// TwinCAT 3 PLC project BROTLibTests
// Title: BROTLibTests
// Company: BROT
// ProjectVersion: 0.1.0
// ProgramVersion: 3.1.4024.66
// libraries:
//   BROTLib, * (BROT)
//   Tc2_MC2, * (Beckhoff Automation GmbH)
//   Tc2_MC2_Drive, * (Beckhoff Automation GmbH)
//   Tc2_NC, * (Beckhoff Automation GmbH)
//   Tc2_Standard, * (Beckhoff Automation GmbH)
//   Tc2_System, * (Beckhoff Automation GmbH)
//   Tc2_Utilities, * (Beckhoff Automation GmbH)
//   Tc3_Module, * (Beckhoff Automation GmbH)
//   TcUnit, * (www.tcunit.org)
// project tree:
//   / PlcTask.TcTTO
//   POUs/ FB_Axis_Tests.TcPOU, FB_Blink_Tests.TcPOU, FB_AstroClockSync_Tests.TcPOU, FB_InfluxLineProtocol_Tests.TcPOU, FB_InfluxMessage_Tests.TcPOU, FB_TelescopeStub.TcPOU, FB_Comm_MQTT_Influx_Tests.TcPOU, FB_BlinkTimingProbe.TcPOU, FB_EscapeInfluxString_Tests.TcPOU, F_SetpointEnableExecute_Tests.TcPOU, FB_InfoConnection_Tests.TcPOU, FB_IsNumericValue_Tests.TcPOU, FB_PointingModel_Tests.TcPOU, FB_Tracking_Tests.TcPOU, FB_YREAL_Tests.TcPOU, MAIN.TcPOU
// real-time tasks:
//   TASK PlcTask: cycle T#10ms, priority 20, ADS port 350

CONFIGURATION BROTLibTests
    RESOURCE PLC ON TwinCAT3
        TASK PlcTask(INTERVAL := T#10ms, PRIORITY := 20);
        PROGRAM MAIN WITH PlcTask : MAIN;
    END_RESOURCE
END_CONFIGURATION

// ---- POUs/MAIN.TcPOU
PROGRAM MAIN
VAR
	// TcUnit finds every FB_TestSuite instance by itself; it is enough to declare them here.
	fbIsNumericValueTests	: FB_IsNumericValue_Tests;
	fbEscapeInfluxTests		: FB_EscapeInfluxString_Tests;
	fbYRealTests			: FB_YREAL_Tests;
	fbTrackingTests			: FB_Tracking_Tests;
	fbPointingModelTests	: FB_PointingModel_Tests;
	fbBlinkTests			: FB_Blink_Tests;
	fbAxisTests				: FB_Axis_Tests;
	fbAstroClockSyncTests	: FB_AstroClockSync_Tests;
	fbInfluxLineProtocolTests	: FB_InfluxLineProtocol_Tests;
	fbInfluxMessageTests		: FB_InfluxMessage_Tests;
	fbCommMqttInfluxTests		: FB_Comm_MQTT_Influx_Tests;
	fbInfoConnectionTests		: FB_InfoConnection_Tests;
	fbSetpointEnableTests		: F_SetpointEnableExecute_Tests;
END_VAR

TcUnit.RUN();

END_PROGRAM

// ---- POUs/FB_IsNumericValue_Tests.TcPOU
// Tests for BROTLib.F_IsNumericValue, which decides whether an Influx field value is written as a number.
FUNCTION_BLOCK FB_IsNumericValue_Tests EXTENDS TcUnit.FB_TestSuite
VAR
END_VAR

Accepts_Plain_Numbers();
Accepts_Signs_And_Exponents();
Rejects_Malformed_Numbers();
Rejects_Non_Numeric_Text();

// Asserts F_IsNumericValue(sValue) = bExpected; the failure message names the offending input.
METHOD PRIVATE Check
VAR_INPUT
	sValue		: STRING(255);
	bExpected	: BOOL;
END_VAR
AssertEquals_BOOL(
	Expected := bExpected,
	Actual := BROTLib.F_IsNumericValue(sValue := sValue),
	Message := CONCAT('F_IsNumericValue on input: ', sValue));
END_METHOD

METHOD PRIVATE Accepts_Plain_Numbers
VAR
	aCases	: ARRAY[1..6] OF STRING(255) := ['0', '15', '15.5', '007', '0.001', '123456789012345678'];
	i		: INT;
END_VAR
TEST('Accepts_Plain_Numbers');
FOR i := 1 TO 6 DO
	Check(sValue := aCases[i], bExpected := TRUE);
END_FOR
TEST_FINISHED();
END_METHOD

METHOD PRIVATE Accepts_Signs_And_Exponents
VAR
	aCases	: ARRAY[1..8] OF STRING(255) := ['-3', '+7', '-0.5', '1e5', '1E-05', '1.0E-5', '-1.5e+3', '2.5E+10'];
	i		: INT;
END_VAR
TEST('Accepts_Signs_And_Exponents');
FOR i := 1 TO 8 DO
	Check(sValue := aCases[i], bExpected := TRUE);
END_FOR
TEST_FINISHED();
END_METHOD

METHOD PRIVATE Rejects_Malformed_Numbers
VAR
	aCases	: ARRAY[1..14] OF STRING(255) := ['', '-', '+', '.', 'e5', '1e', '1e+', '1.5.2', '1e5.5', '--1', '+-1', '1-1', '1e5e5', '1e--5'];
	i		: INT;
END_VAR
TEST('Rejects_Malformed_Numbers');
FOR i := 1 TO 14 DO
	Check(sValue := aCases[i], bExpected := FALSE);
END_FOR
TEST_FINISHED();
END_METHOD

METHOD PRIVATE Rejects_Non_Numeric_Text
VAR
	aCases	: ARRAY[1..9] OF STRING(255) := ['NaN', 'TRUE', 'abc', '12a', '50cm', ' 1', '1 ', '1,5', '0x1F'];
	i		: INT;
END_VAR
TEST('Rejects_Non_Numeric_Text');
FOR i := 1 TO 9 DO
	Check(sValue := aCases[i], bExpected := FALSE);
END_FOR
TEST_FINISHED();
END_METHOD

END_FUNCTION_BLOCK

// ---- POUs/FB_EscapeInfluxString_Tests.TcPOU
// Tests for BROTLib.F_EscapeInfluxString: inside a quoted InfluxDB string field only " and \ need escaping.
FUNCTION_BLOCK FB_EscapeInfluxString_Tests EXTENDS TcUnit.FB_TestSuite
VAR
END_VAR

Leaves_Plain_Text_Unchanged();
Escapes_Double_Quotes();
Escapes_Backslashes();
Doubles_Length_Of_All_Quote_Input();

METHOD PRIVATE Check
VAR_INPUT
	sInput		: STRING(255);
	sExpected	: STRING(255);
END_VAR
AssertEquals_STRING(
	Expected := sExpected,
	Actual := BROTLib.F_EscapeInfluxString(sValue := sInput),
	Message := CONCAT('F_EscapeInfluxString on input: ', sInput));
END_METHOD

METHOD PRIVATE Leaves_Plain_Text_Unchanged
VAR
END_VAR
TEST('Leaves_Plain_Text_Unchanged');
Check(sInput := '', sExpected := '');
Check(sInput := 'plain text', sExpected := 'plain text');
Check(sInput := 'a,b=c d', sExpected := 'a,b=c d');
Check(sInput := 'temp 21.5 C', sExpected := 'temp 21.5 C');
TEST_FINISHED();
END_METHOD

METHOD PRIVATE Escapes_Double_Quotes
VAR
END_VAR
TEST('Escapes_Double_Quotes');
Check(sInput := '"', sExpected := '\"');
Check(sInput := 'say "hi"', sExpected := 'say \"hi\"');
Check(sInput := '""', sExpected := '\"\"');
TEST_FINISHED();
END_METHOD

METHOD PRIVATE Escapes_Backslashes
VAR
END_VAR
TEST('Escapes_Backslashes');
Check(sInput := '\', sExpected := '\\');
Check(sInput := 'C:\temp', sExpected := 'C:\\temp');
// a backslash followed by a quote: both characters are escaped independently
Check(sInput := '\"', sExpected := '\\\"');
TEST_FINISHED();
END_METHOD

METHOD PRIVATE Doubles_Length_Of_All_Quote_Input
VAR
	sInput	: STRING(255);
	sOut	: STRING(255);
	i		: INT;
END_VAR
TEST('Doubles_Length_Of_All_Quote_Input');
sInput := '';
FOR i := 1 TO 100 DO
	sInput := CONCAT(sInput, '"');
END_FOR
sOut := BROTLib.F_EscapeInfluxString(sValue := sInput);
AssertEquals_INT(Expected := 200, Actual := LEN(sOut), Message := '100 quotes must become 100 escaped pairs');
AssertEquals_STRING(Expected := '\"\"', Actual := LEFT(sOut, 4), Message := 'every quote is preceded by one backslash');
TEST_FINISHED();
END_METHOD

END_FUNCTION_BLOCK

// ---- POUs/FB_YREAL_Tests.TcPOU
// Tests for BROTLib.F_YREAL, the linear scaling helper.
FUNCTION_BLOCK FB_YREAL_Tests EXTENDS TcUnit.FB_TestSuite
VAR
END_VAR

Default_Range_Maps_Raw_To_Unit();
Scales_To_Engineering_Range();
Clamps_Unless_Cut_Is_False();
Zero_Width_Input_Range_Returns_Zero();
Inverted_Output_Range_Maps_Correctly();

METHOD PRIVATE CheckNear
VAR_INPUT
	fExpected	: REAL;
	fActual		: REAL;
	fDelta		: REAL;
	sName		: STRING(255);
END_VAR
AssertEquals_REAL(Expected := fExpected, Actual := fActual, Delta := fDelta, Message := sName);
END_METHOD

METHOD PRIVATE Default_Range_Maps_Raw_To_Unit
VAR
END_VAR
TEST('Default_Range_Maps_Raw_To_Unit');
// defaults: 0..32767 -> 0..1
CheckNear(0.0, BROTLib.F_YREAL(fX := 0.0, fXmin := 0.0, fXmax := 32767.0, fYmin := 0.0, fYmax := 1.0, cut := TRUE), 1.0E-6, 'raw 0 -> 0');
CheckNear(1.0, BROTLib.F_YREAL(fX := 32767.0, fXmin := 0.0, fXmax := 32767.0, fYmin := 0.0, fYmax := 1.0, cut := TRUE), 1.0E-6, 'raw 32767 -> 1');
CheckNear(0.5, BROTLib.F_YREAL(fX := 16383.5, fXmin := 0.0, fXmax := 32767.0, fYmin := 0.0, fYmax := 1.0, cut := TRUE), 1.0E-6, 'raw mid-scale -> 0.5');
TEST_FINISHED();
END_METHOD

METHOD PRIVATE Scales_To_Engineering_Range
VAR
END_VAR
TEST('Scales_To_Engineering_Range');
// a 4..20 mA style input
CheckNear(4.0, BROTLib.F_YREAL(fX := 0.0, fXmin := 0.0, fXmax := 32767.0, fYmin := 4.0, fYmax := 20.0, cut := TRUE), 1.0E-5, '4..20: raw 0 -> 4');
CheckNear(20.0, BROTLib.F_YREAL(fX := 32767.0, fXmin := 0.0, fXmax := 32767.0, fYmin := 4.0, fYmax := 20.0, cut := TRUE), 1.0E-5, '4..20: raw 32767 -> 20');
CheckNear(12.0, BROTLib.F_YREAL(fX := 16383.5, fXmin := 0.0, fXmax := 32767.0, fYmin := 4.0, fYmax := 20.0, cut := TRUE), 1.0E-4, '4..20: mid-scale -> 12');
// symmetric ranges on both sides
CheckNear(0.0, BROTLib.F_YREAL(fX := 0.0, fXmin := -10.0, fXmax := 10.0, fYmin := -1.0, fYmax := 1.0, cut := TRUE), 1.0E-6, '-10..10 -> -1..1: 0 -> 0');
CheckNear(0.5, BROTLib.F_YREAL(fX := 5.0, fXmin := -10.0, fXmax := 10.0, fYmin := -1.0, fYmax := 1.0, cut := TRUE), 1.0E-6, '-10..10 -> -1..1: 5 -> 0.5');
CheckNear(-1.0, BROTLib.F_YREAL(fX := -10.0, fXmin := -10.0, fXmax := 10.0, fYmin := -1.0, fYmax := 1.0, cut := TRUE), 1.0E-6, '-10..10 -> -1..1: -10 -> -1');
TEST_FINISHED();
END_METHOD

METHOD PRIVATE Clamps_Unless_Cut_Is_False
VAR
END_VAR
TEST('Clamps_Unless_Cut_Is_False');
// cut defaults to TRUE
CheckNear(1.0, BROTLib.F_YREAL(fX := 40000.0, fXmin := 0.0, fXmax := 32767.0, fYmin := 0.0, fYmax := 1.0, cut := TRUE), 1.0E-6, 'above range is clamped to the maximum');
CheckNear(0.0, BROTLib.F_YREAL(fX := -100.0, fXmin := 0.0, fXmax := 32767.0, fYmin := 0.0, fYmax := 1.0, cut := TRUE), 1.0E-6, 'below range is clamped to the minimum');
CheckNear(20.0, BROTLib.F_YREAL(fX := 40000.0, fXmin := 0.0, fXmax := 32767.0, fYmin := 4.0, fYmax := 20.0, cut := TRUE), 1.0E-5, 'clamping works with an offset range');
// cut = FALSE extrapolates linearly
CheckNear(2.0, BROTLib.F_YREAL(fX := 65534.0, fXmin := 0.0, fXmax := 32767.0, fYmin := 0.0, fYmax := 1.0, cut := FALSE), 1.0E-5, 'unclamped: twice full scale -> 2');
CheckNear(-1.0, BROTLib.F_YREAL(fX := -32767.0, fXmin := 0.0, fXmax := 32767.0, fYmin := 0.0, fYmax := 1.0, cut := FALSE), 1.0E-5, 'unclamped: minus full scale -> -1');
TEST_FINISHED();
END_METHOD

METHOD PRIVATE Zero_Width_Input_Range_Returns_Zero
VAR
END_VAR
TEST('Zero_Width_Input_Range_Returns_Zero');
// fXmax = fXmin would divide by zero; the function guards against it and leaves the result at 0
CheckNear(0.0, BROTLib.F_YREAL(fX := 5.0, fXmin := 1.0, fXmax := 1.0, fYmin := 0.0, fYmax := 1.0, cut := TRUE), 1.0E-6, 'fXmax = fXmin -> 0');
TEST_FINISHED();
END_METHOD

METHOD PRIVATE Inverted_Output_Range_Maps_Correctly
VAR
END_VAR
TEST('Inverted_Output_Range_Maps_Correctly');
// fYmin > fYmax (descending output range); LIMIT needs its low/high bounds the right way round
// regardless of which of fYmin/fYmax is numerically smaller (code review L2, issue #15)
CheckNear(0.75, BROTLib.F_YREAL(fX := 0.25, fXmin := 0.0, fXmax := 1.0, fYmin := 1.0, fYmax := 0.0, cut := TRUE), 1.0E-6, '0.25 on [0,1] -> [1,0]: 0.75');
CheckNear(1.0, BROTLib.F_YREAL(fX := 0.0, fXmin := 0.0, fXmax := 1.0, fYmin := 1.0, fYmax := 0.0, cut := TRUE), 1.0E-6, '0.0 on [0,1] -> [1,0]: 1.0');
CheckNear(0.0, BROTLib.F_YREAL(fX := 1.0, fXmin := 0.0, fXmax := 1.0, fYmin := 1.0, fYmax := 0.0, cut := TRUE), 1.0E-6, '1.0 on [0,1] -> [1,0]: 0.0');
// out-of-range input still clamps to the correct end of the descending range
CheckNear(1.0, BROTLib.F_YREAL(fX := -1.0, fXmin := 0.0, fXmax := 1.0, fYmin := 1.0, fYmax := 0.0, cut := TRUE), 1.0E-6, 'below range clamps to 1.0, not 0.0');
CheckNear(0.0, BROTLib.F_YREAL(fX := 2.0, fXmin := 0.0, fXmax := 1.0, fYmin := 1.0, fYmax := 0.0, cut := TRUE), 1.0E-6, 'above range clamps to 0.0, not 1.0');
TEST_FINISHED();
END_METHOD

END_FUNCTION_BLOCK

// ---- POUs/FB_Tracking_Tests.TcPOU
// Tests for the sidereal tracking functions of BROTLib: F_Azimuthvelocity, F_Elevationvelocity,
// F_Derotatorvelocity and F_DerotatorPosition2.
//
// Two kinds of expected values:
//  * anchors that can be checked by hand (sin/cos of 0, 30, 45, 60, 90 degrees), and
//  * golden values printed by BROTLib/testing/golden_vectors.py, which first validates the same formulas
//    against numerical derivatives of an independent HA/Dec -> Az/El transform (agreement ~4e-10 deg/s).
// All angles are in degrees, velocities in deg/s.
FUNCTION_BLOCK FB_Tracking_Tests EXTENDS TcUnit.FB_TestSuite
VAR CONSTANT
	// Earth's angular rotation rate in deg/s, the same constant as inside the functions
	fOmega		: LREAL := 4.178074605556E-3;
	// Goettingen
	fLat		: LREAL := 51.56;
END_VAR

Elevationvelocity_Anchors();
Azimuthvelocity_Anchors();
Azimuthvelocity_Near_Zenith_Guard();
Derotatorvelocity_Anchors();
DerotatorPosition2_Anchors();
DerotatorPosition2_Stays_In_Range();

METHOD PRIVATE CheckNear
VAR_INPUT
	fExpected	: LREAL;
	fActual		: LREAL;
	fDelta		: LREAL;
	sName		: STRING(255);
END_VAR
AssertEquals_LREAL(Expected := fExpected, Actual := fActual, Delta := fDelta, Message := sName);
END_METHOD

METHOD PRIVATE Elevationvelocity_Anchors
VAR
END_VAR
TEST('Elevationvelocity_Anchors');
CheckNear(0.0, BROTLib.F_Elevationvelocity(azimuth := 0.0, latitude := fLat), 1.0E-15, 'azimuth 0 (north): no elevation rate');
CheckNear(fOmega, BROTLib.F_Elevationvelocity(azimuth := 90.0, latitude := 0.0), 1.0E-15, 'east on the equator: full sidereal rate');
CheckNear(-fOmega, BROTLib.F_Elevationvelocity(azimuth := 270.0, latitude := 0.0), 1.0E-15, 'west on the equator: full rate, falling');
CheckNear(0.5 * fOmega, BROTLib.F_Elevationvelocity(azimuth := 90.0, latitude := 60.0), 1.0E-12, 'east at latitude 60: cos(60) = 0.5');
CheckNear(0.0, BROTLib.F_Elevationvelocity(azimuth := 90.0, latitude := 90.0), 1.0E-12, 'at the pole nothing rises or sets');
CheckNear(0.0021685065117460016, BROTLib.F_Elevationvelocity(azimuth := 123.4, latitude := 51.56), 1.0E-12, 'golden: az 123.4, lat 51.56');
CheckNear(-0.0031335559541669999, BROTLib.F_Elevationvelocity(azimuth := 300.0, latitude := -30.0), 1.0E-12, 'golden: az 300, lat -30');
TEST_FINISHED();
END_METHOD

METHOD PRIVATE Azimuthvelocity_Anchors
VAR
END_VAR
TEST('Azimuthvelocity_Anchors');
CheckNear(0.0032725171421828193, BROTLib.F_Azimuthvelocity(elevation := 0.0, azimuth := 0.0, latitude := 51.56), 1.0E-12, 'golden: horizon, lat 51.56 -> sin(lat) * Omega');
CheckNear(-0.5 * fOmega, BROTLib.F_Azimuthvelocity(elevation := 0.0, azimuth := 100.0, latitude := -30.0), 1.0E-12, 'southern hemisphere: sign flips, sin(-30) = -0.5');
CheckNear(1.4142135623730951 * fOmega, BROTLib.F_Azimuthvelocity(elevation := 45.0, azimuth := 180.0, latitude := 45.0), 1.0E-12, 'south at el 45, lat 45: sqrt(2) * Omega');
CheckNear(0.0, BROTLib.F_Azimuthvelocity(elevation := 45.0, azimuth := 0.0, latitude := 45.0), 1.0E-12, 'north at el 45, lat 45: terms cancel');
CheckNear(0.0046817364334291968, BROTLib.F_Azimuthvelocity(elevation := 30.0, azimuth := 200.0, latitude := 51.56), 1.0E-12, 'golden: el 30, az 200, lat 51.56');
CheckNear(-0.0052225932569449993, BROTLib.F_Azimuthvelocity(elevation := 60.0, azimuth := 300.0, latitude := -30.0), 1.0E-12, 'golden: el 60, az 300, lat -30');
TEST_FINISHED();
END_METHOD

METHOD PRIVATE Azimuthvelocity_Near_Zenith_Guard
VAR
END_VAR
TEST('Azimuthvelocity_Near_Zenith_Guard');
// The formula divides by cos(elevation); below cos = 1e-3 (elevation > 89.943 deg) the function returns 0
// instead of a huge number. The true rate is not 0 there (code review L3); this pins the current behaviour.
CheckNear(0.0, BROTLib.F_Azimuthvelocity(elevation := 90.0, azimuth := 45.0, latitude := 51.56), 0.0, 'zenith: guarded, exactly 0');
CheckNear(0.0, BROTLib.F_Azimuthvelocity(elevation := 89.95, azimuth := 45.0, latitude := 51.56), 0.0, 'el 89.95: inside the guard, exactly 0');
CheckNear(-1.0490784008893366, BROTLib.F_Azimuthvelocity(elevation := 89.9, azimuth := 45.0, latitude := 51.56), 1.0E-9, 'el 89.9: just outside the guard, large but finite');
TEST_FINISHED();
END_METHOD

METHOD PRIVATE Derotatorvelocity_Anchors
VAR
END_VAR
TEST('Derotatorvelocity_Anchors');
CheckNear(-fOmega, BROTLib.F_Derotatorvelocity(elevation := 0.0, azimuth := 0.0, latitude := 0.0, sign := 1.0), 1.0E-15, 'horizon, north, equator: -Omega');
CheckNear(-fOmega, BROTLib.F_Derotatorvelocity(elevation := 0.0, azimuth := 90.0, latitude := 0.0, sign := 1.0), 1.0E-15, 'horizon, east, equator: -Omega');
CheckNear(fOmega, BROTLib.F_Derotatorvelocity(elevation := 0.0, azimuth := 180.0, latitude := 0.0, sign := 1.0), 1.0E-15, 'horizon, south, equator: +Omega');
CheckNear(-2.0 * fOmega, BROTLib.F_Derotatorvelocity(elevation := 60.0, azimuth := 0.0, latitude := 0.0, sign := 1.0), 1.0E-12, 'el 60: 1/cos(60) = 2');
CheckNear(0.0, BROTLib.F_Derotatorvelocity(elevation := 90.0, azimuth := 10.0, latitude := 51.56, sign := 1.0), 0.0, 'zenith: guarded, exactly 0');
CheckNear(0.0037068314748825424, BROTLib.F_Derotatorvelocity(elevation := 30.0, azimuth := 200.0, latitude := 51.56, sign := 1.0), 1.0E-12, 'golden: el 30, az 200, lat 51.56');
CheckNear(-0.00048476279315114428, BROTLib.F_Derotatorvelocity(elevation := 60.0, azimuth := 300.0, latitude := -30.0, sign := 1.0), 1.0E-12, 'golden: el 60, az 300, lat -30');
// sign, added for #16: sign defaults to 1.0 (all the above are unaffected); sign = -1.0 adds twice the
// elevation rate back in, verified against a numerical derivative of F_DerotatorPosition2(..., sign := -1.0)
CheckNear(0.0019300456901029633, BROTLib.F_Derotatorvelocity(elevation := 30.0, azimuth := 200.0, latitude := 51.56, sign := -1.0), 1.0E-12, 'golden: el 30, az 200, lat 51.56, sign -1');
CheckNear(-0.006751874701485144, BROTLib.F_Derotatorvelocity(elevation := 60.0, azimuth := 300.0, latitude := -30.0, sign := -1.0), 1.0E-12, 'golden: el 60, az 300, lat -30, sign -1');
TEST_FINISHED();
END_METHOD

METHOD PRIVATE DerotatorPosition2_Anchors
VAR
END_VAR
TEST('DerotatorPosition2_Anchors');
CheckNear(315.0, BROTLib.F_DerotatorPosition2(azimuth := 90.0, elevation := 0.0, latitude := 45.0, sign := 1.0), 1.0E-9, 'az 90, el 0, lat 45: parallactic angle -45 -> 315');
CheckNear(45.0, BROTLib.F_DerotatorPosition2(azimuth := 270.0, elevation := 0.0, latitude := 45.0, sign := 1.0), 1.0E-9, 'az 270 mirrors az 90: +45');
CheckNear(225.0, BROTLib.F_DerotatorPosition2(azimuth := 90.0, elevation := 45.0, latitude := 0.0, sign := 1.0), 1.0E-9, 'equator, east, el 45: -90 - 45 -> 225');
CheckNear(315.0, BROTLib.F_DerotatorPosition2(azimuth := 90.0, elevation := 45.0, latitude := 0.0, sign := -1.0), 1.0E-9, 'sign -1 adds the elevation instead: -90 + 45 -> 315');
CheckNear(267.36458824003319, BROTLib.F_DerotatorPosition2(azimuth := 123.4, elevation := 56.7, latitude := 51.56, sign := 1.0), 1.0E-9, 'golden: az 123.4, el 56.7, sign +1');
CheckNear(20.764588240033163, BROTLib.F_DerotatorPosition2(azimuth := 123.4, elevation := 56.7, latitude := 51.56, sign := -1.0), 1.0E-9, 'golden: az 123.4, el 56.7, sign -1');
CheckNear(109.48603710615262, BROTLib.F_DerotatorPosition2(azimuth := 300.0, elevation := 20.0, latitude := -30.0, sign := 1.0), 1.0E-9, 'golden: az 300, el 20, lat -30');
// negative azimuth is wrapped into 0..360 before use
CheckNear(15.882548343825519, BROTLib.F_DerotatorPosition2(azimuth := -30.0, elevation := 45.0, latitude := 51.56, sign := 1.0), 1.0E-9, 'golden: az -30 wraps to 330');
CheckNear(BROTLib.F_DerotatorPosition2(azimuth := 330.0, elevation := 45.0, latitude := 51.56, sign := 1.0),
	BROTLib.F_DerotatorPosition2(azimuth := -30.0, elevation := 45.0, latitude := 51.56, sign := 1.0), 1.0E-9, 'az -30 equals az 330');
TEST_FINISHED();
END_METHOD

METHOD PRIVATE DerotatorPosition2_Stays_In_Range
VAR
	aLat		: ARRAY[1..3] OF LREAL := [-60.0, 10.0, 51.56];
	iLat, iAz, iEl	: INT;
	fResult		: LREAL;
	bInRange	: BOOL;
	nChecked	: INT;
END_VAR
TEST('DerotatorPosition2_Stays_In_Range');
// Whatever the pointing direction, the derotator position is a valid angle in [0, 360).
// Azimuths 5, 15, ... 355 avoid the exact ATAN2(0, 0) corner cases; a NaN result also fails the range test.
bInRange := TRUE;
nChecked := 0;
FOR iLat := 1 TO 3 DO
	FOR iAz := 0 TO 35 DO
		FOR iEl := 0 TO 6 DO
			fResult := BROTLib.F_DerotatorPosition2(
				azimuth := 5.0 + 10.0 * iAz,
				elevation := 15.0 * iEl,
				latitude := aLat[iLat],
				sign := 1.0);
			IF NOT (fResult >= 0.0 AND fResult < 360.0) THEN
				bInRange := FALSE;
			END_IF
			nChecked := nChecked + 1;
		END_FOR
	END_FOR
END_FOR
AssertEquals_INT(Expected := 756, Actual := nChecked, Message := 'the whole grid was evaluated');
AssertTrue(Condition := bInRange, Message := 'F_DerotatorPosition2 returned a value outside [0, 360)');
TEST_FINISHED();
END_METHOD

END_FUNCTION_BLOCK

// ---- POUs/FB_PointingModel_Tests.TcPOU
// Tests for BROTLib.FB_PointingModelForward and FB_PointingModelInversion (9-term Tpoint-style model).
//
//   d(az) = AOFF - BNP/cos(el) + AN_A*sin(az)*tan(el) - AE_A*cos(az)*tan(el) + NPAE*tan(el)
//   d(el) = EOFF + AN_E*cos(az) + AE_E*sin(az) + TF*cos(el)
//
// Each term gets its own test at an (az, el) where the expected value follows from sin/cos/tan of 0, 45, 60,
// 90 or 180 degrees. The combined and zenith values come from BROTLib/testing/golden_vectors.py.
FUNCTION_BLOCK FB_PointingModel_Tests EXTENDS TcUnit.FB_TestSuite
VAR
END_VAR

Zero_Coefficients_Give_Zero_Offsets();
AOFF_Is_A_Constant_Azimuth_Offset();
EOFF_Is_A_Constant_Elevation_Offset();
BNP_Scales_With_Secant_Of_Elevation();
NPAE_Scales_With_Tangent_Of_Elevation();
Azimuth_Axis_Tilt_Terms();
Elevation_Terms();
Zenith_Is_Clamped();
Combined_Model_Golden_Vector();
Inversion_Round_Trip();

METHOD PRIVATE CheckNear
VAR_INPUT
	fExpected	: LREAL;
	fActual		: LREAL;
	fDelta		: LREAL;
	sName		: STRING(255);
END_VAR
AssertEquals_LREAL(Expected := fExpected, Actual := fActual, Delta := fDelta, Message := sName);
END_METHOD

METHOD PRIVATE Zero_Coefficients_Give_Zero_Offsets
VAR
	fbModel	: BROTLib.FB_PointingModelForward(AOFF := 0.0, BNP := 0.0, AN_A := 0.0, AE_A := 0.0, NPAE := 0.0, EOFF := 0.0, AN_E := 0.0, AE_E := 0.0, TF := 0.0);
END_VAR
TEST('Zero_Coefficients_Give_Zero_Offsets');
fbModel(fAzimuth := 123.4, fElevation := 45.6);
CheckNear(0.0, fbModel.fAzimuthOffset, 1.0E-15, 'azimuth offset at el 45.6');
CheckNear(0.0, fbModel.fElevationOffset, 1.0E-15, 'elevation offset at el 45.6');
// near the zenith the model divides by cos(el); with all coefficients zero that must still give 0, not NaN
fbModel(fAzimuth := 10.0, fElevation := 90.0);
CheckNear(0.0, fbModel.fAzimuthOffset, 1.0E-15, 'azimuth offset at the zenith');
CheckNear(0.0, fbModel.fElevationOffset, 1.0E-15, 'elevation offset at the zenith');
TEST_FINISHED();
END_METHOD

METHOD PRIVATE AOFF_Is_A_Constant_Azimuth_Offset
VAR
	fbModel	: BROTLib.FB_PointingModelForward(AOFF := 0.25, BNP := 0.0, AN_A := 0.0, AE_A := 0.0, NPAE := 0.0, EOFF := 0.0, AN_E := 0.0, AE_E := 0.0, TF := 0.0);
END_VAR
TEST('AOFF_Is_A_Constant_Azimuth_Offset');
fbModel(fAzimuth := 10.0, fElevation := 20.0);
CheckNear(0.25, fbModel.fAzimuthOffset, 1.0E-12, 'azimuth offset at az 10, el 20');
CheckNear(0.0, fbModel.fElevationOffset, 1.0E-15, 'elevation is not affected');
fbModel(fAzimuth := 250.0, fElevation := 70.0);
CheckNear(0.25, fbModel.fAzimuthOffset, 1.0E-12, 'same offset at az 250, el 70');
TEST_FINISHED();
END_METHOD

METHOD PRIVATE EOFF_Is_A_Constant_Elevation_Offset
VAR
	fbModel	: BROTLib.FB_PointingModelForward(AOFF := 0.0, BNP := 0.0, AN_A := 0.0, AE_A := 0.0, NPAE := 0.0, EOFF := -0.125, AN_E := 0.0, AE_E := 0.0, TF := 0.0);
END_VAR
TEST('EOFF_Is_A_Constant_Elevation_Offset');
fbModel(fAzimuth := 10.0, fElevation := 20.0);
CheckNear(-0.125, fbModel.fElevationOffset, 1.0E-12, 'elevation offset at az 10, el 20');
CheckNear(0.0, fbModel.fAzimuthOffset, 1.0E-15, 'azimuth is not affected');
fbModel(fAzimuth := 250.0, fElevation := 70.0);
CheckNear(-0.125, fbModel.fElevationOffset, 1.0E-12, 'same offset at az 250, el 70');
TEST_FINISHED();
END_METHOD

METHOD PRIVATE BNP_Scales_With_Secant_Of_Elevation
VAR
	fbModel	: BROTLib.FB_PointingModelForward(AOFF := 0.0, BNP := 0.01, AN_A := 0.0, AE_A := 0.0, NPAE := 0.0, EOFF := 0.0, AN_E := 0.0, AE_E := 0.0, TF := 0.0);
END_VAR
TEST('BNP_Scales_With_Secant_Of_Elevation');
fbModel(fAzimuth := 37.0, fElevation := 0.0);
CheckNear(-0.01, fbModel.fAzimuthOffset, 1.0E-12, 'el 0: -BNP / cos(0)');
fbModel(fAzimuth := 37.0, fElevation := 60.0);
CheckNear(-0.02, fbModel.fAzimuthOffset, 1.0E-12, 'el 60: -BNP / 0.5');
CheckNear(0.0, fbModel.fElevationOffset, 1.0E-15, 'elevation is not affected');
TEST_FINISHED();
END_METHOD

METHOD PRIVATE NPAE_Scales_With_Tangent_Of_Elevation
VAR
	fbModel	: BROTLib.FB_PointingModelForward(AOFF := 0.0, BNP := 0.0, AN_A := 0.0, AE_A := 0.0, NPAE := 0.01, EOFF := 0.0, AN_E := 0.0, AE_E := 0.0, TF := 0.0);
END_VAR
TEST('NPAE_Scales_With_Tangent_Of_Elevation');
fbModel(fAzimuth := 37.0, fElevation := 0.0);
CheckNear(0.0, fbModel.fAzimuthOffset, 1.0E-15, 'el 0: NPAE * tan(0)');
fbModel(fAzimuth := 37.0, fElevation := 45.0);
CheckNear(0.01, fbModel.fAzimuthOffset, 1.0E-12, 'el 45: NPAE * tan(45)');
TEST_FINISHED();
END_METHOD

METHOD PRIVATE Azimuth_Axis_Tilt_Terms
VAR
	fbNorthSouth	: BROTLib.FB_PointingModelForward(AOFF := 0.0, BNP := 0.0, AN_A := 0.02, AE_A := 0.0, NPAE := 0.0, EOFF := 0.0, AN_E := 0.0, AE_E := 0.0, TF := 0.0);
	fbEastWest		: BROTLib.FB_PointingModelForward(AOFF := 0.0, BNP := 0.0, AN_A := 0.0, AE_A := 0.03, NPAE := 0.0, EOFF := 0.0, AN_E := 0.0, AE_E := 0.0, TF := 0.0);
END_VAR
TEST('Azimuth_Axis_Tilt_Terms');
// AN_A * sin(az) * tan(el): largest towards east/west
fbNorthSouth(fAzimuth := 90.0, fElevation := 45.0);
CheckNear(0.02, fbNorthSouth.fAzimuthOffset, 1.0E-12, 'AN_A at az 90, el 45');
fbNorthSouth(fAzimuth := 0.0, fElevation := 45.0);
CheckNear(0.0, fbNorthSouth.fAzimuthOffset, 1.0E-12, 'AN_A vanishes at az 0');
fbNorthSouth(fAzimuth := 270.0, fElevation := 45.0);
CheckNear(-0.02, fbNorthSouth.fAzimuthOffset, 1.0E-12, 'AN_A changes sign at az 270');
// -AE_A * cos(az) * tan(el): largest towards north/south, with a leading minus
fbEastWest(fAzimuth := 180.0, fElevation := 45.0);
CheckNear(0.03, fbEastWest.fAzimuthOffset, 1.0E-12, 'AE_A at az 180, el 45');
fbEastWest(fAzimuth := 0.0, fElevation := 45.0);
CheckNear(-0.03, fbEastWest.fAzimuthOffset, 1.0E-12, 'AE_A at az 0, el 45');
fbEastWest(fAzimuth := 90.0, fElevation := 45.0);
CheckNear(0.0, fbEastWest.fAzimuthOffset, 1.0E-12, 'AE_A vanishes at az 90');
TEST_FINISHED();
END_METHOD

METHOD PRIVATE Elevation_Terms
VAR
	fbAnE	: BROTLib.FB_PointingModelForward(AOFF := 0.0, BNP := 0.0, AN_A := 0.0, AE_A := 0.0, NPAE := 0.0, EOFF := 0.0, AN_E := 0.04, AE_E := 0.0, TF := 0.0);
	fbAeE	: BROTLib.FB_PointingModelForward(AOFF := 0.0, BNP := 0.0, AN_A := 0.0, AE_A := 0.0, NPAE := 0.0, EOFF := 0.0, AN_E := 0.0, AE_E := 0.05, TF := 0.0);
	fbTF	: BROTLib.FB_PointingModelForward(AOFF := 0.0, BNP := 0.0, AN_A := 0.0, AE_A := 0.0, NPAE := 0.0, EOFF := 0.0, AN_E := 0.0, AE_E := 0.0, TF := 0.06);
END_VAR
TEST('Elevation_Terms');
// AN_E * cos(az)
fbAnE(fAzimuth := 0.0, fElevation := 30.0);
CheckNear(0.04, fbAnE.fElevationOffset, 1.0E-12, 'AN_E at az 0');
fbAnE(fAzimuth := 90.0, fElevation := 30.0);
CheckNear(0.0, fbAnE.fElevationOffset, 1.0E-12, 'AN_E vanishes at az 90');
// AE_E * sin(az)
fbAeE(fAzimuth := 90.0, fElevation := 30.0);
CheckNear(0.05, fbAeE.fElevationOffset, 1.0E-12, 'AE_E at az 90');
fbAeE(fAzimuth := 0.0, fElevation := 30.0);
CheckNear(0.0, fbAeE.fElevationOffset, 1.0E-12, 'AE_E vanishes at az 0');
// TF * cos(el): gravitational flexure, largest at the horizon
fbTF(fAzimuth := 200.0, fElevation := 0.0);
CheckNear(0.06, fbTF.fElevationOffset, 1.0E-12, 'TF at the horizon');
fbTF(fAzimuth := 200.0, fElevation := 60.0);
CheckNear(0.03, fbTF.fElevationOffset, 1.0E-12, 'TF at el 60: cos(60) = 0.5');
fbTF(fAzimuth := 200.0, fElevation := 90.0);
CheckNear(0.0, fbTF.fElevationOffset, 1.0E-12, 'TF vanishes at the zenith');
TEST_FINISHED();
END_METHOD

METHOD PRIVATE Zenith_Is_Clamped
VAR
	fbNpae	: BROTLib.FB_PointingModelForward(AOFF := 0.0, BNP := 0.0, AN_A := 0.0, AE_A := 0.0, NPAE := 0.001, EOFF := 0.0, AN_E := 0.0, AE_E := 0.0, TF := 0.0);
	fbBnp	: BROTLib.FB_PointingModelForward(AOFF := 0.0, BNP := 0.001, AN_A := 0.0, AE_A := 0.0, NPAE := 0.0, EOFF := 0.0, AN_E := 0.0, AE_E := 0.0, TF := 0.0);
END_VAR
TEST('Zenith_Is_Clamped');
// From el = 89.9 the model uses fixed tan = 572.957... and cos = 0.001745... so that it never divides by ~0.
fbNpae(fAzimuth := 10.0, fElevation := 89.95);
CheckNear(0.57295721335430339, fbNpae.fAzimuthOffset, 1.0E-9, 'NPAE at el 89.95 uses the clamped tangent');
fbBnp(fAzimuth := 10.0, fElevation := 89.95);
CheckNear(-0.57295808601915088, fbBnp.fAzimuthOffset, 1.0E-9, 'BNP at el 89.95 uses the clamped cosine');
fbBnp(fAzimuth := 10.0, fElevation := 90.0);
CheckNear(-0.57295808601915088, fbBnp.fAzimuthOffset, 1.0E-9, 'BNP at el 90 gives the same clamped value');
TEST_FINISHED();
END_METHOD

METHOD PRIVATE Combined_Model_Golden_Vector
VAR
	fbModel	: BROTLib.FB_PointingModelForward(
				AOFF := 0.1, BNP := 0.02, AN_A := 0.03, AE_A := -0.04, NPAE := 0.05,
				EOFF := -0.06, AN_E := 0.07, AE_E := -0.08, TF := 0.09);
END_VAR
TEST('Combined_Model_Golden_Vector');
fbModel(fAzimuth := 123.4, fElevation := 56.7);
CheckNear(0.14429632570655807, fbModel.fAzimuthOffset, 1.0E-12, 'azimuth offset with all nine terms');
CheckNear(-0.11590942724719037, fbModel.fElevationOffset, 1.0E-12, 'elevation offset with all nine terms');
TEST_FINISHED();
END_METHOD

METHOD PRIVATE Inversion_Round_Trip
VAR
	fbModel		: BROTLib.FB_PointingModelForward(
					AOFF := 0.1, BNP := 0.02, AN_A := 0.03, AE_A := -0.04, NPAE := 0.05,
					EOFF := -0.06, AN_E := 0.07, AE_E := -0.08, TF := 0.09);
	fbInverse	: BROTLib.FB_PointingModelInversion(fbPointing := fbModel);
	aAz			: ARRAY[1..4] OF LREAL := [15.0, 100.0, 200.0, 330.0];
	aEl			: ARRAY[1..3] OF LREAL := [10.0, 45.0, 80.0];
	iAz, iEl	: INT;
	fdAz, fdEl	: LREAL;
END_VAR
TEST('Inversion_Round_Trip');
// The inversion solves d = model(pos - d) by fixed-point iteration. So evaluating the forward model at the
// corrected position must give back exactly the offsets the inversion reported.
FOR iAz := 1 TO 4 DO
	FOR iEl := 1 TO 3 DO
		fbInverse(fAzimuth := aAz[iAz], fElevation := aEl[iEl]);
		fdAz := fbInverse.fAzimuthOffset;
		fdEl := fbInverse.fElevationOffset;
		fbModel(fAzimuth := aAz[iAz] - fdAz, fElevation := aEl[iEl] - fdEl);
		CheckNear(fdAz, fbModel.fAzimuthOffset, 1.0E-9, 'azimuth offset is a fixed point of the model');
		CheckNear(fdEl, fbModel.fElevationOffset, 1.0E-9, 'elevation offset is a fixed point of the model');
	END_FOR
END_FOR
// and the offsets are non-trivial, so the loop above is not comparing zeros
fbInverse(fAzimuth := 100.0, fElevation := 45.0);
AssertTrue(Condition := ABS(fbInverse.fAzimuthOffset) > 0.01, Message := 'inversion returned a non-trivial azimuth offset');
TEST_FINISHED();
END_METHOD

END_FUNCTION_BLOCK

// ---- POUs/FB_Blink_Tests.TcPOU
// Tests for BROTLib.FB_BLINK (lamp/indicator flasher built from two TOF timers).
//
// The single-cycle tests check the mode logic. Timing_Follows_Mode runs all four blink modes side by side for
// about a second and compares the measured high/low durations with a simulation of the exact TOF chain
// (BROTLib/testing/check_blink_horn.py): at a 10 ms task cycle the steady state is ON + 10 ms high and
// OFF + 20 ms low. The tolerance covers task jitter, which is larger on the user-mode runtime.
//
// FB_Horn is not covered here: it now shares FB_BLINK's exact IMPULS/PAUSE oscillator (fixed in #14) but
// has its own test suite scope if one is added later; see BROTLib/testing/check_blink_horn.py's horn().
FUNCTION_BLOCK FB_Blink_Tests EXTENDS TcUnit.FB_TestSuite
VAR
	fbProbeSlow		: FB_BlinkTimingProbe;
	fbProbeFast		: FB_BlinkTimingProbe;
	fbProbeShort	: FB_BlinkTimingProbe;
	fbProbeLong		: FB_BlinkTimingProbe;
	bTimingChecked	: BOOL;
END_VAR
VAR CONSTANT
	tTolerance		: TIME := T#60MS;
END_VAR

Off_And_On_Modes();
Mode_Selects_On_And_Off_Times();
Blink_Modes_Start_High();
Timing_Follows_Mode();

// Asserts that tActual is within tTolerance of tExpected; the failure message shows the measured value.
METHOD PRIVATE CheckTime
VAR_INPUT
	tExpected	: TIME;
	tActual		: TIME;
	sName		: STRING(255);
END_VAR
AssertTrue(
	Condition := (tActual + tTolerance >= tExpected) AND (tActual <= tExpected + tTolerance),
	Message := CONCAT(CONCAT(sName, ': measured '), TIME_TO_STRING(tActual)));
END_METHOD

METHOD PRIVATE Off_And_On_Modes
VAR
	fbOff	: BROTLib.FB_BLINK;
	fbOn	: BROTLib.FB_BLINK;
END_VAR
TEST('Off_And_On_Modes');
fbOff(blink := BROTLib.E_Blink.off);
fbOn(blink := BROTLib.E_Blink.on);
AssertFalse(Condition := fbOff.Q, Message := 'off: Q is FALSE');
AssertTrue(Condition := fbOn.Q, Message := 'on: Q is TRUE');
TEST_FINISHED();
END_METHOD

METHOD PRIVATE Mode_Selects_On_And_Off_Times
VAR
	fbSlow, fbFast, fbShort, fbLong	: BROTLib.FB_BLINK;
END_VAR
TEST('Mode_Selects_On_And_Off_Times');
fbSlow(blink := BROTLib.E_Blink.slow);
fbFast(blink := BROTLib.E_Blink.fast);
fbShort(blink := BROTLib.E_Blink.short);
fbLong(blink := BROTLib.E_Blink.long);
AssertEquals_TIME(Expected := T#500MS, Actual := fbSlow.ON_TIME, Message := 'slow: ON_TIME');
AssertEquals_TIME(Expected := T#500MS, Actual := fbSlow.OFF_TIME, Message := 'slow: OFF_TIME');
AssertEquals_TIME(Expected := T#250MS, Actual := fbFast.ON_TIME, Message := 'fast: ON_TIME');
AssertEquals_TIME(Expected := T#250MS, Actual := fbFast.OFF_TIME, Message := 'fast: OFF_TIME');
AssertEquals_TIME(Expected := T#100MS, Actual := fbShort.ON_TIME, Message := 'short: ON_TIME');
AssertEquals_TIME(Expected := T#900MS, Actual := fbShort.OFF_TIME, Message := 'short: OFF_TIME');
AssertEquals_TIME(Expected := T#900MS, Actual := fbLong.ON_TIME, Message := 'long: ON_TIME');
AssertEquals_TIME(Expected := T#100MS, Actual := fbLong.OFF_TIME, Message := 'long: OFF_TIME');
TEST_FINISHED();
END_METHOD

METHOD PRIVATE Blink_Modes_Start_High
VAR
	fbSlow, fbFast, fbShort, fbLong	: BROTLib.FB_BLINK;
END_VAR
TEST('Blink_Modes_Start_High');
fbSlow(blink := BROTLib.E_Blink.slow);
fbFast(blink := BROTLib.E_Blink.fast);
fbShort(blink := BROTLib.E_Blink.short);
fbLong(blink := BROTLib.E_Blink.long);
AssertTrue(Condition := fbSlow.Q, Message := 'slow: Q is TRUE on the first call');
AssertTrue(Condition := fbFast.Q, Message := 'fast: Q is TRUE on the first call');
AssertTrue(Condition := fbShort.Q, Message := 'short: Q is TRUE on the first call');
AssertTrue(Condition := fbLong.Q, Message := 'long: Q is TRUE on the first call');
TEST_FINISHED();
END_METHOD

METHOD PRIVATE Timing_Follows_Mode
VAR
END_VAR
TEST('Timing_Follows_Mode');
// this test spans many PLC cycles: the probes run every cycle and are evaluated once they are all done
fbProbeSlow(eMode := BROTLib.E_Blink.slow);
fbProbeFast(eMode := BROTLib.E_Blink.fast);
fbProbeShort(eMode := BROTLib.E_Blink.short);
fbProbeLong(eMode := BROTLib.E_Blink.long);

IF fbProbeSlow.bDone AND fbProbeFast.bDone AND fbProbeShort.bDone AND fbProbeLong.bDone AND NOT bTimingChecked THEN
	bTimingChecked := TRUE;
	AssertFalse(Condition := fbProbeSlow.bTimedOut OR fbProbeFast.bTimedOut OR fbProbeShort.bTimedOut OR fbProbeLong.bTimedOut,
		Message := 'every mode completed one high/low period within 4 s');

	CheckTime(T#510MS, fbProbeSlow.tHigh, 'slow: high time');
	CheckTime(T#520MS, fbProbeSlow.tLow, 'slow: low time');
	CheckTime(T#260MS, fbProbeFast.tHigh, 'fast: high time');
	CheckTime(T#270MS, fbProbeFast.tLow, 'fast: low time');
	CheckTime(T#110MS, fbProbeShort.tHigh, 'short: high time');
	CheckTime(T#920MS, fbProbeShort.tLow, 'short: low time');
	CheckTime(T#910MS, fbProbeLong.tHigh, 'long: high time');
	CheckTime(T#120MS, fbProbeLong.tLow, 'long: low time');
	TEST_FINISHED();
END_IF
END_METHOD

END_FUNCTION_BLOCK

// ---- POUs/FB_BlinkTimingProbe.TcPOU
// Test helper: drives one FB_BLINK in the given mode and measures, in real time, how long Q stays high after the
// first call (tHigh) and how long it then stays low (tLow). Call it every cycle; bDone is set when both are known,
// or when nothing happened within tTimeout (bTimedOut).
FUNCTION_BLOCK FB_BlinkTimingProbe
VAR_INPUT
	eMode		: BROTLib.E_Blink;
END_VAR
VAR_OUTPUT
	bDone		: BOOL;
	bTimedOut	: BOOL;
	tHigh		: TIME;
	tLow		: TIME;
END_VAR
VAR
	fbBlink		: BROTLib.FB_BLINK;
	nState		: INT := 0;
	tStart		: TIME;
	tEdge		: TIME;
END_VAR
VAR CONSTANT
	tTimeout	: TIME := T#4S;
END_VAR

IF bDone THEN
	RETURN;
END_IF

fbBlink(blink := eMode);

CASE nState OF
	0:	// first call: Q is high from here on
		tStart := TIME();
		nState := 1;
	1:	// wait for the falling edge
		IF NOT fbBlink.Q THEN
			tEdge := TIME();
			tHigh := tEdge - tStart;
			nState := 2;
		END_IF
	2:	// wait for the next rising edge
		IF fbBlink.Q THEN
			tLow := TIME() - tEdge;
			bDone := TRUE;
		END_IF
END_CASE

IF NOT bDone AND (TIME() - tStart) > tTimeout THEN
	bTimedOut := TRUE;
	bDone := TRUE;
END_IF

END_FUNCTION_BLOCK

// ---- POUs/FB_Axis_Tests.TcPOU
// Tests for the parts of FB_Axis that do not need a real NC axis: the AXIS_REF is a plain local structure with
// no NC behind it, so the MC_* blocks report errors and never confirm a command. What can be checked is what
// FB_Axis computes itself: the actual position (plain and modulo), isTracking, and that homing/move requests are
// kept or ignored as intended. Homing completion (Homed) and the setpoint generator need the NC and are covered
// by the hardware checks, not here.
// Each test calls the block twice because ActualPosition is read at the end of a cycle and used in the next.
FUNCTION_BLOCK FB_Axis_Tests EXTENDS TcUnit.FB_TestSuite

ActualPosition_Reads_ActPos();
ActualPosition_Modulo_Reads_ModuloActPos();
IsTracking_Envelope();
IsTracking_Requires_Tracking();
IsTracking_Modulo_Wrap_Known_Limitation();
Move_Is_Ignored_Without_Calibration();
Home_Request_Is_Kept_While_Not_Homed();

// AXIS_REF is a function block whose NcToPlc is not writable from outside; a pointer sidesteps that.
METHOD PRIVATE SetActPos
VAR_INPUT
	fValue	: LREAL;
END_VAR
VAR_IN_OUT
	axisRef	: AXIS_REF;
END_VAR
VAR
	pValue	: POINTER TO LREAL;
END_VAR
pValue := ADR(axisRef.NcToPlc.ActPos);
pValue^ := fValue;
END_METHOD

// AXIS_REF is a function block whose NcToPlc is not writable from outside; a pointer sidesteps that.
METHOD PRIVATE SetModuloActPos
VAR_INPUT
	fValue	: LREAL;
END_VAR
VAR_IN_OUT
	axisRef	: AXIS_REF;
END_VAR
VAR
	pValue	: POINTER TO LREAL;
END_VAR
pValue := ADR(axisRef.NcToPlc.ModuloActPos);
pValue^ := fValue;
END_METHOD

METHOD PRIVATE ActualPosition_Reads_ActPos
VAR
	fbAxis	: FB_Axis;
	axisRef	: AXIS_REF;
END_VAR
TEST('ActualPosition_Reads_ActPos');
SetActPos(axisRef := axisRef, fValue := 123.456);
SetModuloActPos(axisRef := axisRef, fValue := 7.0);
fbAxis(AxisRef := axisRef);
AssertEquals_LREAL(Expected := 123.456, Actual := fbAxis.ActualPosition, Delta := 1.0E-12, Message := 'plain axis reports ActPos');
TEST_FINISHED();
END_METHOD

METHOD PRIVATE ActualPosition_Modulo_Reads_ModuloActPos
VAR
	fbAxis	: FB_Axis;
	axisRef	: AXIS_REF;
END_VAR
TEST('ActualPosition_Modulo_Reads_ModuloActPos');
SetActPos(axisRef := axisRef, fValue := 725.0);
SetModuloActPos(axisRef := axisRef, fValue := 5.0);
fbAxis.isModuloAxis := TRUE;
fbAxis(AxisRef := axisRef);
AssertEquals_LREAL(Expected := 5.0, Actual := fbAxis.ActualPosition, Delta := 1.0E-12, Message := 'modulo axis reports ModuloActPos');
TEST_FINISHED();
END_METHOD

METHOD PRIVATE IsTracking_Envelope
VAR
	fbAxis	: FB_Axis;
	axisRef	: AXIS_REF;
END_VAR
TEST('IsTracking_Envelope');
fbAxis.Tracking := TRUE;
fbAxis.Position := 10.0;
fbAxis.TrackEnvelope := 5.0;	// arcsec

SetActPos(axisRef := axisRef, fValue := 10.0 + 4.0 / 3600.0);
fbAxis(AxisRef := axisRef);
fbAxis(AxisRef := axisRef);
AssertTrue(Condition := fbAxis.isTracking, Message := '4 arcsec off, envelope 5 arcsec: tracking');

SetActPos(axisRef := axisRef, fValue := 10.0 - 6.0 / 3600.0);
fbAxis(AxisRef := axisRef);
fbAxis(AxisRef := axisRef);
AssertFalse(Condition := fbAxis.isTracking, Message := '6 arcsec off, envelope 5 arcsec: not tracking');
TEST_FINISHED();
END_METHOD

METHOD PRIVATE IsTracking_Requires_Tracking
VAR
	fbAxis	: FB_Axis;
	axisRef	: AXIS_REF;
END_VAR
TEST('IsTracking_Requires_Tracking');
fbAxis.Tracking := FALSE;
fbAxis.Position := 10.0;
SetActPos(axisRef := axisRef, fValue := 10.0);
fbAxis(AxisRef := axisRef);
fbAxis(AxisRef := axisRef);
AssertFalse(Condition := fbAxis.isTracking, Message := 'on position but tracking not requested');
TEST_FINISHED();
END_METHOD

METHOD PRIVATE IsTracking_Modulo_Wrap_Known_Limitation
VAR
	fbAxis	: FB_Axis;
	axisRef	: AXIS_REF;
END_VAR
TEST('IsTracking_Modulo_Wrap_Known_Limitation');
// Pins the CURRENT behaviour: the position difference is not wrapped on a modulo axis, so 0.001 deg
// against 359.999 deg (0.002 deg apart on the circle) is not seen as tracking. Flip the assertion when
// FB_Axis handles the wrap.
fbAxis.isModuloAxis := TRUE;
fbAxis.Tracking := TRUE;
fbAxis.Position := 0.001;
fbAxis.TrackEnvelope := 10.0;	// arcsec, 0.002 deg = 7.2 arcsec is inside
SetModuloActPos(axisRef := axisRef, fValue := 359.999);
fbAxis(AxisRef := axisRef);
fbAxis(AxisRef := axisRef);
AssertFalse(Condition := fbAxis.isTracking, Message := 'modulo wrap is not handled (known limitation)');
TEST_FINISHED();
END_METHOD

METHOD PRIVATE Move_Is_Ignored_Without_Calibration
VAR
	fbAxis	: FB_Axis;
	axisRef	: AXIS_REF;
END_VAR
TEST('Move_Is_Ignored_Without_Calibration');
fbAxis.MoveAxis := TRUE;
fbAxis.Position := 50.0;
fbAxis(AxisRef := axisRef);
fbAxis(AxisRef := axisRef);
AssertFalse(Condition := fbAxis.Calibrated, Message := 'a fresh axis is not calibrated');
AssertFalse(Condition := fbAxis.MoveDone, Message := 'no move without calibration');
AssertTrue(Condition := fbAxis.MoveAxis, Message := 'the request is kept, not consumed');
TEST_FINISHED();
END_METHOD

METHOD PRIVATE Home_Request_Is_Kept_While_Not_Homed
VAR
	fbAxis	: FB_Axis;
	axisRef	: AXIS_REF;
END_VAR
TEST('Home_Request_Is_Kept_While_Not_Homed');
fbAxis.HomeAxis := TRUE;
fbAxis(AxisRef := axisRef);
fbAxis(AxisRef := axisRef);
AssertFalse(Condition := fbAxis.Calibrated, Message := 'not calibrated without Homed');
AssertFalse(Condition := fbAxis.HomeDone, Message := 'HomeDone is low while not homed');
AssertTrue(Condition := fbAxis.HomeAxis, Message := 'the home request stays set until the axis is homed');
TEST_FINISHED();
END_METHOD

END_FUNCTION_BLOCK

// ---- POUs/FB_AstroClockSync_Tests.TcPOU
// Tests for BROTLib.FB_AstroClockSync, the sync and validity logic of FB_AstroClock (BROTLib issue #3).
//
// Every test drives the Busy and Err inputs the way NT_GetTime does: Busy is TRUE while the ADS read runs, and
// falls in the same cycle in which Err rises when the read fails. No ADS and no timers are involved, so all
// tests finish within a single call.
FUNCTION_BLOCK FB_AstroClockSync_Tests EXTENDS TcUnit.FB_TestSuite

Invalid_Before_First_Read();
Successful_Read_Synchronizes_Once();
Failed_Read_Does_Not_Synchronize();
Error_Held_While_Idle_Is_Counted_Once();
Recovers_After_Failed_First_Read();
Valid_Survives_Transient_Errors();
Stays_Valid_After_Many_Errors();
Success_Resets_Error_Count();

METHOD PRIVATE Invalid_Before_First_Read
VAR
	fbSync	: BROTLib.FB_AstroClockSync;
END_VAR
TEST('Invalid_Before_First_Read');
fbSync(bBusy := FALSE, bError := FALSE);
AssertFalse(Condition := fbSync.bValid, Message := 'idle: not valid');
AssertFalse(Condition := fbSync.bSynchronize, Message := 'idle: no sync');
// read in progress: still nothing to trust
fbSync(bBusy := TRUE, bError := FALSE);
AssertFalse(Condition := fbSync.bValid, Message := 'busy: not valid');
AssertFalse(Condition := fbSync.bSynchronize, Message := 'busy: no sync');
TEST_FINISHED();
END_METHOD

METHOD PRIVATE Successful_Read_Synchronizes_Once
VAR
	fbSync	: BROTLib.FB_AstroClockSync;
END_VAR
TEST('Successful_Read_Synchronizes_Once');
fbSync(bBusy := TRUE, bError := FALSE);
AssertFalse(Condition := fbSync.bSynchronize, Message := 'while busy: no sync yet');
fbSync(bBusy := FALSE, bError := FALSE);
AssertTrue(Condition := fbSync.bSynchronize, Message := 'busy fell without error: sync');
AssertTrue(Condition := fbSync.bValid, Message := 'busy fell without error: valid');
AssertEquals_UINT(Expected := 0, Actual := fbSync.nErrors, Message := 'no errors');
fbSync(bBusy := FALSE, bError := FALSE);
AssertFalse(Condition := fbSync.bSynchronize, Message := 'sync is a one-cycle pulse');
AssertTrue(Condition := fbSync.bValid, Message := 'stays valid');
TEST_FINISHED();
END_METHOD

METHOD PRIVATE Failed_Read_Does_Not_Synchronize
VAR
	fbSync	: BROTLib.FB_AstroClockSync;
END_VAR
TEST('Failed_Read_Does_Not_Synchronize');
// this is the original bug: Busy falls while Err rises, and the stale time struct was loaded into the RTCs
fbSync(bBusy := TRUE, bError := FALSE);
fbSync(bBusy := FALSE, bError := TRUE);
AssertFalse(Condition := fbSync.bSynchronize, Message := 'failed read: no sync');
AssertFalse(Condition := fbSync.bValid, Message := 'failed first read: not valid');
AssertEquals_UINT(Expected := 1, Actual := fbSync.nErrors, Message := 'one error counted');
TEST_FINISHED();
END_METHOD

METHOD PRIVATE Error_Held_While_Idle_Is_Counted_Once
VAR
	fbSync	: BROTLib.FB_AstroClockSync;
	i		: INT;
END_VAR
TEST('Error_Held_While_Idle_Is_Counted_Once');
// NT_GetTime keeps Err TRUE until the next start; that must not count as new errors or new syncs
fbSync(bBusy := TRUE, bError := FALSE);
fbSync(bBusy := FALSE, bError := TRUE);
FOR i := 1 TO 10 DO
	fbSync(bBusy := FALSE, bError := TRUE);
	AssertFalse(Condition := fbSync.bSynchronize, Message := 'idle with Err held: no sync');
END_FOR
AssertEquals_UINT(Expected := 1, Actual := fbSync.nErrors, Message := 'still one error');
TEST_FINISHED();
END_METHOD

METHOD PRIVATE Recovers_After_Failed_First_Read
VAR
	fbSync	: BROTLib.FB_AstroClockSync;
END_VAR
TEST('Recovers_After_Failed_First_Read');
fbSync(bBusy := TRUE, bError := FALSE);
fbSync(bBusy := FALSE, bError := TRUE);
// next read: the start clears Err, the read succeeds
fbSync(bBusy := TRUE, bError := FALSE);
fbSync(bBusy := FALSE, bError := FALSE);
AssertTrue(Condition := fbSync.bSynchronize, Message := 'second read: sync');
AssertTrue(Condition := fbSync.bValid, Message := 'second read: valid');
AssertEquals_UINT(Expected := 0, Actual := fbSync.nErrors, Message := 'error count cleared');
TEST_FINISHED();
END_METHOD

METHOD PRIVATE Valid_Survives_Transient_Errors
VAR
	fbSync	: BROTLib.FB_AstroClockSync;
END_VAR
TEST('Valid_Survives_Transient_Errors');
// the RTC keeps counting: failed reads after a good one only make the last sync older
fbSync(bBusy := TRUE, bError := FALSE);
fbSync(bBusy := FALSE, bError := FALSE);
fbSync(bBusy := TRUE, bError := FALSE);
fbSync(bBusy := FALSE, bError := TRUE);
fbSync(bBusy := TRUE, bError := FALSE);
fbSync(bBusy := FALSE, bError := TRUE);
AssertFalse(Condition := fbSync.bSynchronize, Message := 'failed reads do not sync');
AssertTrue(Condition := fbSync.bValid, Message := 'still valid after 2 errors');
AssertEquals_UINT(Expected := 2, Actual := fbSync.nErrors, Message := 'two errors counted');
TEST_FINISHED();
END_METHOD

METHOD PRIVATE Stays_Valid_After_Many_Errors
VAR
	fbSync	: BROTLib.FB_AstroClockSync;
	i		: INT;
END_VAR
TEST('Stays_Valid_After_Many_Errors');
fbSync(bBusy := TRUE, bError := FALSE);
fbSync(bBusy := FALSE, bError := FALSE);
FOR i := 1 TO 20 DO
	fbSync(bBusy := TRUE, bError := FALSE);
	fbSync(bBusy := FALSE, bError := TRUE);
	AssertFalse(Condition := fbSync.bSynchronize, Message := 'failed read: no sync');
END_FOR
// a long outage must not invalidate the time: the RTC is still counting
AssertTrue(Condition := fbSync.bValid, Message := 'still valid after 20 errors in a row');
AssertEquals_UINT(Expected := 20, Actual := fbSync.nErrors, Message := 'twenty errors counted');
TEST_FINISHED();
END_METHOD

METHOD PRIVATE Success_Resets_Error_Count
VAR
	fbSync	: BROTLib.FB_AstroClockSync;
	i		: INT;
END_VAR
TEST('Success_Resets_Error_Count');
fbSync(bBusy := TRUE, bError := FALSE);
fbSync(bBusy := FALSE, bError := FALSE);
FOR i := 1 TO 3 DO
	fbSync(bBusy := TRUE, bError := FALSE);
	fbSync(bBusy := FALSE, bError := TRUE);
END_FOR
// the link comes back after some failures
fbSync(bBusy := TRUE, bError := FALSE);
fbSync(bBusy := FALSE, bError := FALSE);
AssertTrue(Condition := fbSync.bSynchronize, Message := 'sync after recovery');
AssertTrue(Condition := fbSync.bValid, Message := 'valid');
AssertEquals_UINT(Expected := 0, Actual := fbSync.nErrors, Message := 'error count cleared');
TEST_FINISHED();
END_METHOD

END_FUNCTION_BLOCK

// ---- POUs/FB_InfluxLineProtocol_Tests.TcPOU
// Tests for the InfluxDB line protocol helpers behind FB_Comm_MQTT_Influx.Publish / PublishLog (BROTLib issue #4):
// F_InfluxFieldValue (integer / float / boolean / quoted string), F_EscapeInfluxTag (tag values, field keys, measurement
// names), F_TruncateInfluxEscaped (cut an escaped string without splitting an escape pair) and F_InfluxTimestamp
// (FILETIME to unix ns, #38).
FUNCTION_BLOCK FB_InfluxLineProtocol_Tests EXTENDS TcUnit.FB_TestSuite

Integers_Get_Trailing_i();
Decimals_Stay_Floats();
Exponents_Are_Floats_Not_Integers();
Booleans_Are_Not_Quoted();
Text_Is_Quoted_And_Escaped();
Near_Numbers_Are_Text();
Tag_Plain_Text_Unchanged();
Tag_Escapes_Space_Comma_And_Equals();
Measurement_Name_Keeps_Equals();
Truncate_Leaves_Short_Input();
Truncate_Cuts_Plain_Text();
Truncate_Does_Not_Split_Escape_Pairs();
Timestamp_Unix_Epoch_Is_Zero();
Timestamp_Known_Date();
Timestamp_Keeps_100ns_Resolution();
Timestamp_Before_1970_Is_Empty();

METHOD PRIVATE CheckValue
VAR_INPUT
	sInput		: STRING(255);
	sExpected	: STRING(255);
END_VAR
AssertEquals_STRING(
	Expected := sExpected,
	Actual := BROTLib.F_InfluxFieldValue(sValue := sInput),
	Message := CONCAT('F_InfluxFieldValue on input: ', sInput));
END_METHOD

METHOD PRIVATE CheckTag
VAR_INPUT
	sInput		: STRING(255);
	bEquals		: BOOL;
	sExpected	: STRING(255);
END_VAR
AssertEquals_STRING(
	Expected := sExpected,
	Actual := BROTLib.F_EscapeInfluxTag(sValue := sInput, bEscapeEquals := bEquals),
	Message := CONCAT('F_EscapeInfluxTag on input: ', sInput));
END_METHOD

METHOD PRIVATE CheckTruncate
VAR_INPUT
	sInput		: STRING(255);
	nMax		: INT;
	sExpected	: STRING(255);
END_VAR
AssertEquals_STRING(
	Expected := sExpected,
	Actual := BROTLib.F_TruncateInfluxEscaped(sEscaped := sInput, nMaxLen := nMax),
	Message := CONCAT('F_TruncateInfluxEscaped on input: ', sInput));
END_METHOD

METHOD PRIVATE Integers_Get_Trailing_i
VAR
END_VAR
TEST('Integers_Get_Trailing_i');
CheckValue(sInput := '15', sExpected := '15i');
CheckValue(sInput := '0', sExpected := '0i');
CheckValue(sInput := '-3', sExpected := '-3i');
CheckValue(sInput := '+7', sExpected := '+7i');
TEST_FINISHED();
END_METHOD

METHOD PRIVATE Decimals_Stay_Floats
VAR
END_VAR
TEST('Decimals_Stay_Floats');
CheckValue(sInput := '15.5', sExpected := '15.5');
CheckValue(sInput := '-0.25', sExpected := '-0.25');
CheckValue(sInput := '15.0', sExpected := '15.0');
TEST_FINISHED();
END_METHOD

METHOD PRIVATE Exponents_Are_Floats_Not_Integers
VAR
END_VAR
TEST('Exponents_Are_Floats_Not_Integers');
// 1e5 has no '.', but '1e5i' is invalid line protocol (BROTLib issue #4)
CheckValue(sInput := '1e5', sExpected := '1e5');
CheckValue(sInput := '1E-05', sExpected := '1E-05');
CheckValue(sInput := '2.5e3', sExpected := '2.5e3');
CheckValue(sInput := '-4e+2', sExpected := '-4e+2');
TEST_FINISHED();
END_METHOD

METHOD PRIVATE Booleans_Are_Not_Quoted
VAR
END_VAR
TEST('Booleans_Are_Not_Quoted');
CheckValue(sInput := 'TRUE', sExpected := 'TRUE');
CheckValue(sInput := 'false', sExpected := 'false');
TEST_FINISHED();
END_METHOD

METHOD PRIVATE Text_Is_Quoted_And_Escaped
VAR
END_VAR
TEST('Text_Is_Quoted_And_Escaped');
CheckValue(sInput := 'abc', sExpected := '"abc"');
CheckValue(sInput := '', sExpected := '""');
CheckValue(sInput := 'say "hi"', sExpected := '"say \"hi\""');
TEST_FINISHED();
END_METHOD

METHOD PRIVATE Near_Numbers_Are_Text
VAR
END_VAR
TEST('Near_Numbers_Are_Text');
CheckValue(sInput := '1e', sExpected := '"1e"');
CheckValue(sInput := '12abc', sExpected := '"12abc"');
CheckValue(sInput := 'NaN', sExpected := '"NaN"');
CheckValue(sInput := '1.2.3', sExpected := '"1.2.3"');
TEST_FINISHED();
END_METHOD

METHOD PRIVATE Tag_Plain_Text_Unchanged
VAR
END_VAR
TEST('Tag_Plain_Text_Unchanged');
CheckTag(sInput := '', bEquals := TRUE, sExpected := '');
CheckTag(sInput := 'CX-4E6032', bEquals := TRUE, sExpected := 'CX-4E6032');
CheckTag(sInput := 'environment', bEquals := FALSE, sExpected := 'environment');
TEST_FINISHED();
END_METHOD

METHOD PRIVATE Tag_Escapes_Space_Comma_And_Equals
VAR
END_VAR
TEST('Tag_Escapes_Space_Comma_And_Equals');
CheckTag(sInput := 'CX 4E', bEquals := TRUE, sExpected := 'CX\ 4E');
CheckTag(sInput := 'a,b', bEquals := TRUE, sExpected := 'a\,b');
CheckTag(sInput := 'k=v', bEquals := TRUE, sExpected := 'k\=v');
CheckTag(sInput := 'CX 4E,60=32', bEquals := TRUE, sExpected := 'CX\ 4E\,60\=32');
TEST_FINISHED();
END_METHOD

METHOD PRIVATE Measurement_Name_Keeps_Equals
VAR
END_VAR
TEST('Measurement_Name_Keeps_Equals');
// a measurement name only needs its space and comma escaped
CheckTag(sInput := 'a=b c,d', bEquals := FALSE, sExpected := 'a=b\ c\,d');
TEST_FINISHED();
END_METHOD

METHOD PRIVATE Truncate_Leaves_Short_Input
VAR
END_VAR
TEST('Truncate_Leaves_Short_Input');
CheckTruncate(sInput := 'abc', nMax := 3, sExpected := 'abc');
CheckTruncate(sInput := 'abc', nMax := 10, sExpected := 'abc');
CheckTruncate(sInput := '', nMax := 5, sExpected := '');
TEST_FINISHED();
END_METHOD

METHOD PRIVATE Truncate_Cuts_Plain_Text
VAR
END_VAR
TEST('Truncate_Cuts_Plain_Text');
CheckTruncate(sInput := 'abcdef', nMax := 4, sExpected := 'abcd');
CheckTruncate(sInput := 'abcdef', nMax := 0, sExpected := '');
CheckTruncate(sInput := 'abcdef', nMax := -2, sExpected := '');
TEST_FINISHED();
END_METHOD

METHOD PRIVATE Truncate_Does_Not_Split_Escape_Pairs
VAR
END_VAR
TEST('Truncate_Does_Not_Split_Escape_Pairs');
// a lone trailing backslash would escape the closing quote of the string field
CheckTruncate(sInput := 'ab\"cd', nMax := 3, sExpected := 'ab');
CheckTruncate(sInput := 'ab\"cd', nMax := 4, sExpected := 'ab\"');
CheckTruncate(sInput := 'a\\b', nMax := 2, sExpected := 'a');
CheckTruncate(sInput := 'a\\b', nMax := 3, sExpected := 'a\\');
// three backslashes: an escaped backslash and the start of an escaped quote
CheckTruncate(sInput := 'x\\\"y', nMax := 4, sExpected := 'x\\');
TEST_FINISHED();
END_METHOD

METHOD PRIVATE CheckTimestamp
VAR_INPUT
	nFileTime	: ULINT;
	sExpected	: STRING(255);
END_VAR
AssertEquals_STRING(
	Expected := sExpected,
	Actual := BROTLib.F_InfluxTimestamp(nFileTime := nFileTime),
	Message := CONCAT('F_InfluxTimestamp on FILETIME: ', ULINT_TO_STRING(nFileTime)));
END_METHOD

METHOD PRIVATE Timestamp_Unix_Epoch_Is_Zero
VAR
END_VAR
TEST('Timestamp_Unix_Epoch_Is_Zero');
// 1970-01-01 00:00:00 UTC as FILETIME (100 ns since 1601-01-01)
CheckTimestamp(nFileTime := 116444736000000000, sExpected := '0');
TEST_FINISHED();
END_METHOD

METHOD PRIVATE Timestamp_Known_Date
VAR
END_VAR
TEST('Timestamp_Known_Date');
// 2026-10-08 12:34:56 UTC = unix 1791462896 s
CheckTimestamp(nFileTime := 134359364960000000, sExpected := '1791462896000000000');
TEST_FINISHED();
END_METHOD

METHOD PRIVATE Timestamp_Keeps_100ns_Resolution
VAR
END_VAR
TEST('Timestamp_Keeps_100ns_Resolution');
CheckTimestamp(nFileTime := 116444736000000001, sExpected := '100');
CheckTimestamp(nFileTime := 116444736012345678, sExpected := '1234567800');
TEST_FINISHED();
END_METHOD

METHOD PRIVATE Timestamp_Before_1970_Is_Empty
VAR
END_VAR
TEST('Timestamp_Before_1970_Is_Empty');
// an unset clock: no timestamp, the receiver stamps the line
CheckTimestamp(nFileTime := 0, sExpected := '');
CheckTimestamp(nFileTime := 116444735999999999, sExpected := '');
TEST_FINISHED();
END_METHOD

END_FUNCTION_BLOCK

// ---- POUs/FB_InfluxMessage_Tests.TcPOU
// Tests for BROTLib.FB_InfluxMessage, the parser of incoming MQTT command payloads
// (measurement[,tags] parameter=value[,parameter=value ...] [timestamp]). Since BROTLib#39 it returns the first pair
// and a 'remaining' payload for the next one; the first five cases are the behaviour it had before and still has.
FUNCTION_BLOCK FB_InfluxMessage_Tests EXTENDS TcUnit.FB_TestSuite
VAR
END_VAR

Single_Pair();
Numbers_Keep_Sign_And_Exponent();
Tags_Are_Dropped();
Trailing_Timestamp_Is_Dropped();
Quoted_String_Value_Loses_Quotes();
Several_Pairs_Walk_Via_Remaining();
Remaining_Keeps_Tags_And_Timestamp();
No_Space_Gives_Empty_Outputs();
Outputs_Are_Reset_Between_Calls();

// Parses sPayload with a fresh instance (method locals are re-initialised on every call) and asserts all four outputs;
// the failure message names the payload.
METHOD PRIVATE Check
VAR_INPUT
	sPayload		: STRING(255);
	sMeasurement	: STRING(255);
	sParameter		: STRING(255);
	sValue			: STRING(255);
	sRemaining		: STRING(255);
END_VAR
VAR
	fb				: BROTLib.FB_InfluxMessage;
END_VAR
fb(sPayload := sPayload);
AssertEquals_STRING(Expected := sMeasurement, Actual := fb.measurement, Message := CONCAT('measurement of: ', sPayload));
AssertEquals_STRING(Expected := sParameter, Actual := fb.parameter, Message := CONCAT('parameter of: ', sPayload));
AssertEquals_STRING(Expected := sValue, Actual := fb.value, Message := CONCAT('value of: ', sPayload));
AssertEquals_STRING(Expected := sRemaining, Actual := fb.remaining, Message := CONCAT('remaining of: ', sPayload));
END_METHOD

METHOD PRIVATE Single_Pair
VAR
END_VAR
TEST('Single_Pair');
Check(sPayload := 'command park=1', sMeasurement := 'command', sParameter := 'park', sValue := '1', sRemaining := '');
Check(sPayload := 'command track=1', sMeasurement := 'command', sParameter := 'track', sValue := '1', sRemaining := '');
TEST_FINISHED();
END_METHOD

METHOD PRIVATE Numbers_Keep_Sign_And_Exponent
VAR
END_VAR
TEST('Numbers_Keep_Sign_And_Exponent');
Check(sPayload := 'command rightascension=123.456', sMeasurement := 'command', sParameter := 'rightascension', sValue := '123.456', sRemaining := '');
Check(sPayload := 'command declination=-56.7', sMeasurement := 'command', sParameter := 'declination', sValue := '-56.7', sRemaining := '');
Check(sPayload := 'command offset=1.5E-3', sMeasurement := 'command', sParameter := 'offset', sValue := '1.5E-3', sRemaining := '');
TEST_FINISHED();
END_METHOD

// Tags after the measurement are accepted but not returned.
METHOD PRIVATE Tags_Are_Dropped
VAR
END_VAR
TEST('Tags_Are_Dropped');
Check(sPayload := 'command,site=a park=1', sMeasurement := 'command', sParameter := 'park', sValue := '1', sRemaining := '');
TEST_FINISHED();
END_METHOD

METHOD PRIVATE Trailing_Timestamp_Is_Dropped
VAR
END_VAR
TEST('Trailing_Timestamp_Is_Dropped');
Check(sPayload := 'command park=1 1700000000000000000', sMeasurement := 'command', sParameter := 'park', sValue := '1', sRemaining := '');
Check(sPayload := 'command,site=a track=1 1700000000000000000', sMeasurement := 'command', sParameter := 'track', sValue := '1', sRemaining := '');
TEST_FINISHED();
END_METHOD

// The surrounding quotes of an Influx string value are stripped.
METHOD PRIVATE Quoted_String_Value_Loses_Quotes
VAR
END_VAR
TEST('Quoted_String_Value_Loses_Quotes');
Check(sPayload := 'command name="abc"', sMeasurement := 'command', sParameter := 'name', sValue := 'abc', sRemaining := '');
TEST_FINISHED();
END_METHOD

// BROTLib#39: the first pair is returned and 'remaining' is a complete payload for the next one; feeding it back in
// walks the whole field set.
METHOD PRIVATE Several_Pairs_Walk_Via_Remaining
VAR
END_VAR
TEST('Several_Pairs_Walk_Via_Remaining');
Check(sPayload := 'command a=1,b=2,c=3', sMeasurement := 'command', sParameter := 'a', sValue := '1', sRemaining := 'command b=2,c=3');
Check(sPayload := 'command b=2,c=3', sMeasurement := 'command', sParameter := 'b', sValue := '2', sRemaining := 'command c=3');
Check(sPayload := 'command c=3', sMeasurement := 'command', sParameter := 'c', sValue := '3', sRemaining := '');
TEST_FINISHED();
END_METHOD

// The tags stay in front and the timestamp stays at the end; it is dropped from the value of the last pair.
METHOD PRIVATE Remaining_Keeps_Tags_And_Timestamp
VAR
END_VAR
TEST('Remaining_Keeps_Tags_And_Timestamp');
Check(sPayload := 'command,site=x a=1,b=2 1700000000000000000', sMeasurement := 'command', sParameter := 'a', sValue := '1', sRemaining := 'command,site=x b=2 1700000000000000000');
Check(sPayload := 'command,site=x b=2 1700000000000000000', sMeasurement := 'command', sParameter := 'b', sValue := '2', sRemaining := '');
TEST_FINISHED();
END_METHOD

// Without a space there is no field set: the block returns early and every output stays empty.
METHOD PRIVATE No_Space_Gives_Empty_Outputs
VAR
END_VAR
TEST('No_Space_Gives_Empty_Outputs');
Check(sPayload := 'command', sMeasurement := '', sParameter := '', sValue := '', sRemaining := '');
Check(sPayload := '', sMeasurement := '', sParameter := '', sValue := '', sRemaining := '');
TEST_FINISHED();
END_METHOD

METHOD PRIVATE Outputs_Are_Reset_Between_Calls
VAR
	fb	: BROTLib.FB_InfluxMessage;
END_VAR
TEST('Outputs_Are_Reset_Between_Calls');
// a caller that reuses the instance (the multi-field loop does) must never see the previous pair again
fb(sPayload := 'command a=1,b=2');
AssertEquals_STRING(Expected := 'a', Actual := fb.parameter, Message := 'first call returns a');
fb(sPayload := 'command');
AssertEquals_STRING(Expected := '', Actual := fb.measurement, Message := 'measurement is reset');
AssertEquals_STRING(Expected := '', Actual := fb.parameter, Message := 'parameter is reset');
AssertEquals_STRING(Expected := '', Actual := fb.value, Message := 'value is reset');
AssertEquals_STRING(Expected := '', Actual := fb.remaining, Message := 'remaining is reset');
TEST_FINISHED();
END_METHOD

END_FUNCTION_BLOCK

// ---- POUs/FB_Comm_MQTT_Influx_Tests.TcPOU
// Tests for the command dispatch of BROTLib.FB_Comm_MQTT_Influx (BROTLib#39): single-field messages as pyBROT and
// BROTgui send them, and multi-field messages where track/slew must see the data of the same message. The handler is
// called directly with a payload; no MQTT connection is made. A stub records what it asks the telescope to do.
FUNCTION_BLOCK FB_Comm_MQTT_Influx_Tests EXTENDS TcUnit.FB_TestSuite
VAR
	fbComm	: BROTLib.FB_Comm_MQTT_Influx;
	stub	: FB_TelescopeStub;
	bReady	: BOOL;
	bSingle_Field_Messages_Still_Fill_The_Buffer	: BOOL;
	bData_Before_Verb_In_One_Message	: BOOL;
	bVerb_First_Uses_Data_From_The_Same_Message	: BOOL;
	bSame_Message_Data_Beats_The_Buffer	: BOOL;
	bIncomplete_Pair_Is_Dropped	: BOOL;
	bBuffer_Is_Cleared_After_Track	: BOOL;
	bSlew_Takes_Elevation_And_Azimuth_From_One_Message	: BOOL;
	bTrailing_Timestamp_Does_Not_Break_The_Last_Field	: BOOL;
	bOther_Measurement_Is_Ignored	: BOOL;
	bFields_Beyond_The_Eighth_Are_Ignored	: BOOL;
	bNon_Numeric_Coordinate_Is_Rejected	: BOOL;
	bOut_Of_Range_Coordinates_Are_Rejected	: BOOL;
	bRange_Limits_Are_Accepted	: BOOL;
	bRejected_Value_Clears_The_Buffer	: BOOL;
END_VAR

IF NOT bReady THEN
	bReady := TRUE;
	fbComm.Telescope := stub;
END_IF
Single_Field_Messages_Still_Fill_The_Buffer();
Data_Before_Verb_In_One_Message();
Verb_First_Uses_Data_From_The_Same_Message();
Same_Message_Data_Beats_The_Buffer();
Incomplete_Pair_Is_Dropped();
Buffer_Is_Cleared_After_Track();
Slew_Takes_Elevation_And_Azimuth_From_One_Message();
Trailing_Timestamp_Does_Not_Break_The_Last_Field();
Other_Measurement_Is_Ignored();
Fields_Beyond_The_Eighth_Are_Ignored();
Non_Numeric_Coordinate_Is_Rejected();
Out_Of_Range_Coordinates_Are_Rejected();
Range_Limits_Are_Accepted();
Rejected_Value_Clears_The_Buffer();

// Puts the handler and the stub back to a clean state; every test runs its body once.
METHOD PRIVATE ResetHandler
VAR_INPUT
END_VAR
// drain whatever the previous test left in the handler's buffers: track and slew consume and clear them
fbComm._handleMQTTMessage(sPayloadRcv := 'command track=1');
fbComm._handleMQTTMessage(sPayloadRcv := 'command slew=1');
stub.ClearCounters();
END_METHOD

// The way pyBROT and BROTgui send it today: three messages, the buffer is consumed by track.
METHOD PRIVATE Single_Field_Messages_Still_Fill_The_Buffer
VAR
END_VAR
TEST('Single_Field_Messages_Still_Fill_The_Buffer');
IF NOT bSingle_Field_Messages_Still_Fill_The_Buffer THEN
	bSingle_Field_Messages_Still_Fill_The_Buffer := TRUE;
	ResetHandler();
	fbComm._handleMQTTMessage(sPayloadRcv := 'command rightascension=10.5');
	fbComm._handleMQTTMessage(sPayloadRcv := 'command declination=20.5');
	AssertEquals_INT(Expected := 0, Actual := stub.nTrack, Message := 'before track: number of Track calls');
	fbComm._handleMQTTMessage(sPayloadRcv := 'command track=1');
	AssertEquals_INT(Expected := 1, Actual := stub.nTrack, Message := 'after track: number of Track calls');
	AssertEquals_LREAL(Expected := 10.5, Actual := stub.fTrackRa, Delta := 1.0E-9, Message := 'after track: right ascension');
	AssertEquals_LREAL(Expected := 20.5, Actual := stub.fTrackDec, Delta := 1.0E-9, Message := 'after track: declination');
	TEST_FINISHED();
END_IF
END_METHOD

METHOD PRIVATE Data_Before_Verb_In_One_Message
VAR
END_VAR
TEST('Data_Before_Verb_In_One_Message');
IF NOT bData_Before_Verb_In_One_Message THEN
	bData_Before_Verb_In_One_Message := TRUE;
	ResetHandler();
	fbComm._handleMQTTMessage(sPayloadRcv := 'command rightascension=10.5,declination=20.5,track=1');
	AssertEquals_INT(Expected := 1, Actual := stub.nTrack, Message := 'one message: number of Track calls');
	AssertEquals_LREAL(Expected := 10.5, Actual := stub.fTrackRa, Delta := 1.0E-9, Message := 'one message: right ascension');
	AssertEquals_LREAL(Expected := 20.5, Actual := stub.fTrackDec, Delta := 1.0E-9, Message := 'one message: declination');
	TEST_FINISHED();
END_IF
END_METHOD

// The data pass runs before the verb pass, so the field order does not matter.
METHOD PRIVATE Verb_First_Uses_Data_From_The_Same_Message
VAR
END_VAR
TEST('Verb_First_Uses_Data_From_The_Same_Message');
IF NOT bVerb_First_Uses_Data_From_The_Same_Message THEN
	bVerb_First_Uses_Data_From_The_Same_Message := TRUE;
	ResetHandler();
	fbComm._handleMQTTMessage(sPayloadRcv := 'command track=1,rightascension=10.5,declination=20.5');
	AssertEquals_INT(Expected := 1, Actual := stub.nTrack, Message := 'verb first: number of Track calls');
	AssertEquals_LREAL(Expected := 10.5, Actual := stub.fTrackRa, Delta := 1.0E-9, Message := 'verb first: right ascension');
	AssertEquals_LREAL(Expected := 20.5, Actual := stub.fTrackDec, Delta := 1.0E-9, Message := 'verb first: declination');
	TEST_FINISHED();
END_IF
END_METHOD

// An old buffer value must never be combined with the new target.
METHOD PRIVATE Same_Message_Data_Beats_The_Buffer
VAR
END_VAR
TEST('Same_Message_Data_Beats_The_Buffer');
IF NOT bSame_Message_Data_Beats_The_Buffer THEN
	bSame_Message_Data_Beats_The_Buffer := TRUE;
	ResetHandler();
	fbComm._handleMQTTMessage(sPayloadRcv := 'command rightascension=1.5');
	fbComm._handleMQTTMessage(sPayloadRcv := 'command declination=2.5');
	fbComm._handleMQTTMessage(sPayloadRcv := 'command rightascension=10.5,declination=20.5,track=1');
	AssertEquals_INT(Expected := 1, Actual := stub.nTrack, Message := 'stale buffer: number of Track calls');
	AssertEquals_LREAL(Expected := 10.5, Actual := stub.fTrackRa, Delta := 1.0E-9, Message := 'stale buffer: right ascension');
	AssertEquals_LREAL(Expected := 20.5, Actual := stub.fTrackDec, Delta := 1.0E-9, Message := 'stale buffer: declination');
	TEST_FINISHED();
END_IF
END_METHOD

// Same as the buffered form: no declination, no Track call.
METHOD PRIVATE Incomplete_Pair_Is_Dropped
VAR
END_VAR
TEST('Incomplete_Pair_Is_Dropped');
IF NOT bIncomplete_Pair_Is_Dropped THEN
	bIncomplete_Pair_Is_Dropped := TRUE;
	ResetHandler();
	fbComm._handleMQTTMessage(sPayloadRcv := 'command rightascension=10.5,track=1');
	AssertEquals_INT(Expected := 0, Actual := stub.nTrack, Message := 'declination missing: number of Track calls');
	TEST_FINISHED();
END_IF
END_METHOD

// The second track finds an empty buffer and is dropped, the first call stays the last one.
METHOD PRIVATE Buffer_Is_Cleared_After_Track
VAR
END_VAR
TEST('Buffer_Is_Cleared_After_Track');
IF NOT bBuffer_Is_Cleared_After_Track THEN
	bBuffer_Is_Cleared_After_Track := TRUE;
	ResetHandler();
	fbComm._handleMQTTMessage(sPayloadRcv := 'command rightascension=10.5,declination=20.5,track=1');
	fbComm._handleMQTTMessage(sPayloadRcv := 'command track=1');
	AssertEquals_INT(Expected := 1, Actual := stub.nTrack, Message := 'second track without data: number of Track calls');
	AssertEquals_LREAL(Expected := 10.5, Actual := stub.fTrackRa, Delta := 1.0E-9, Message := 'second track without data: right ascension');
	AssertEquals_LREAL(Expected := 20.5, Actual := stub.fTrackDec, Delta := 1.0E-9, Message := 'second track without data: declination');
	TEST_FINISHED();
END_IF
END_METHOD

METHOD PRIVATE Slew_Takes_Elevation_And_Azimuth_From_One_Message
VAR
END_VAR
TEST('Slew_Takes_Elevation_And_Azimuth_From_One_Message');
IF NOT bSlew_Takes_Elevation_And_Azimuth_From_One_Message THEN
	bSlew_Takes_Elevation_And_Azimuth_From_One_Message := TRUE;
	ResetHandler();
	fbComm._handleMQTTMessage(sPayloadRcv := 'command slew=1,azimuth=120.5,elevation=45.5');
	AssertEquals_INT(Expected := 1, Actual := stub.nSlew, Message := 'slew: number of Slew calls');
	AssertEquals_LREAL(Expected := 120.5, Actual := stub.fSlewAz, Delta := 1.0E-9, Message := 'slew: azimuth');
	AssertEquals_LREAL(Expected := 45.5, Actual := stub.fSlewAlt, Delta := 1.0E-9, Message := 'slew: altitude');
	TEST_FINISHED();
END_IF
END_METHOD

METHOD PRIVATE Trailing_Timestamp_Does_Not_Break_The_Last_Field
VAR
END_VAR
TEST('Trailing_Timestamp_Does_Not_Break_The_Last_Field');
IF NOT bTrailing_Timestamp_Does_Not_Break_The_Last_Field THEN
	bTrailing_Timestamp_Does_Not_Break_The_Last_Field := TRUE;
	ResetHandler();
	fbComm._handleMQTTMessage(sPayloadRcv := 'command rightascension=10.5,declination=20.5,track=1 1700000000000000000');
	AssertEquals_INT(Expected := 1, Actual := stub.nTrack, Message := 'timestamp: number of Track calls');
	AssertEquals_LREAL(Expected := 10.5, Actual := stub.fTrackRa, Delta := 1.0E-9, Message := 'timestamp: right ascension');
	AssertEquals_LREAL(Expected := 20.5, Actual := stub.fTrackDec, Delta := 1.0E-9, Message := 'timestamp: declination');
	TEST_FINISHED();
END_IF
END_METHOD

METHOD PRIVATE Other_Measurement_Is_Ignored
VAR
END_VAR
TEST('Other_Measurement_Is_Ignored');
IF NOT bOther_Measurement_Is_Ignored THEN
	bOther_Measurement_Is_Ignored := TRUE;
	ResetHandler();
	fbComm._handleMQTTMessage(sPayloadRcv := 'status rightascension=10.5,declination=20.5,track=1');
	AssertEquals_INT(Expected := 0, Actual := stub.nTrack, Message := 'measurement status: number of Track calls');
	TEST_FINISHED();
END_IF
END_METHOD

// At most 8 fields per message (a malformed message must not spin the scan cycle); the rest is logged and ignored.
METHOD PRIVATE Fields_Beyond_The_Eighth_Are_Ignored
VAR
END_VAR
TEST('Fields_Beyond_The_Eighth_Are_Ignored');
IF NOT bFields_Beyond_The_Eighth_Are_Ignored THEN
	bFields_Beyond_The_Eighth_Are_Ignored := TRUE;
	ResetHandler();
	fbComm._handleMQTTMessage(sPayloadRcv := 'command rightascension=10.5,declination=20.5,x1=0,x2=0,x3=0,x4=0,x5=0,x6=0,track=1');
	AssertEquals_INT(Expected := 0, Actual := stub.nTrack, Message := 'track is the ninth field: number of Track calls');
	TEST_FINISHED();
END_IF
END_METHOD

// STRING_TO_LREAL turns garbage into 0.0, a valid coordinate; it must not reach Track (#27).
METHOD PRIVATE Non_Numeric_Coordinate_Is_Rejected
VAR
END_VAR
TEST('Non_Numeric_Coordinate_Is_Rejected');
IF NOT bNon_Numeric_Coordinate_Is_Rejected THEN
	bNon_Numeric_Coordinate_Is_Rejected := TRUE;
	ResetHandler();
	fbComm._handleMQTTMessage(sPayloadRcv := 'command rightascension=abc,declination=20.5,track=1');
	AssertEquals_INT(Expected := 0, Actual := stub.nTrack, Message := 'rightascension=abc: number of Track calls');
	fbComm._handleMQTTMessage(sPayloadRcv := 'command rightascension=10.5,declination=nan,track=1');
	AssertEquals_INT(Expected := 0, Actual := stub.nTrack, Message := 'declination=nan: number of Track calls');
	TEST_FINISHED();
END_IF
END_METHOD

METHOD PRIVATE Out_Of_Range_Coordinates_Are_Rejected
VAR
END_VAR
TEST('Out_Of_Range_Coordinates_Are_Rejected');
IF NOT bOut_Of_Range_Coordinates_Are_Rejected THEN
	bOut_Of_Range_Coordinates_Are_Rejected := TRUE;
	ResetHandler();
	fbComm._handleMQTTMessage(sPayloadRcv := 'command rightascension=10.5,declination=95,track=1');
	AssertEquals_INT(Expected := 0, Actual := stub.nTrack, Message := 'declination=95: number of Track calls');
	fbComm._handleMQTTMessage(sPayloadRcv := 'command rightascension=1e999,declination=20.5,track=1');
	AssertEquals_INT(Expected := 0, Actual := stub.nTrack, Message := 'rightascension=1e999: number of Track calls');
	fbComm._handleMQTTMessage(sPayloadRcv := 'command elevation=120,azimuth=10,slew=1');
	AssertEquals_INT(Expected := 0, Actual := stub.nSlew, Message := 'elevation=120: number of Slew calls');
	TEST_FINISHED();
END_IF
END_METHOD

// The limits themselves are valid values; so are signs and exponents.
METHOD PRIVATE Range_Limits_Are_Accepted
VAR
END_VAR
TEST('Range_Limits_Are_Accepted');
IF NOT bRange_Limits_Are_Accepted THEN
	bRange_Limits_Are_Accepted := TRUE;
	ResetHandler();
	fbComm._handleMQTTMessage(sPayloadRcv := 'command rightascension=0,declination=-90,track=1');
	AssertEquals_INT(Expected := 1, Actual := stub.nTrack, Message := 'ra=0, dec=-90: number of Track calls');
	fbComm._handleMQTTMessage(sPayloadRcv := 'command rightascension=360,declination=+9e1,track=1');
	AssertEquals_INT(Expected := 2, Actual := stub.nTrack, Message := 'ra=360, dec=+9e1: number of Track calls');
	AssertEquals_LREAL(Expected := 90.0, Actual := stub.fTrackDec, Delta := 1.0E-9, Message := 'dec=+9e1: declination');
	TEST_FINISHED();
END_IF
END_METHOD

// A rejected coordinate must not fall back to one buffered by an earlier message: the track is dropped instead.
METHOD PRIVATE Rejected_Value_Clears_The_Buffer
VAR
END_VAR
TEST('Rejected_Value_Clears_The_Buffer');
IF NOT bRejected_Value_Clears_The_Buffer THEN
	bRejected_Value_Clears_The_Buffer := TRUE;
	ResetHandler();
	fbComm._handleMQTTMessage(sPayloadRcv := 'command rightascension=1.5');
	fbComm._handleMQTTMessage(sPayloadRcv := 'command rightascension=abc,declination=20.5,track=1');
	AssertEquals_INT(Expected := 0, Actual := stub.nTrack, Message := 'buffered ra, then ra=abc: number of Track calls');
	TEST_FINISHED();
END_IF
END_METHOD

END_FUNCTION_BLOCK

// ---- POUs/FB_TelescopeStub.TcPOU
// Minimal I_Telescope that only records what the MQTT handler asks it to do.
FUNCTION_BLOCK FB_TelescopeStub IMPLEMENTS BROTLib.I_Telescope
VAR_OUTPUT
	nTrack			: INT;		// number of Track() calls
	fTrackRa		: LREAL;	// arguments of the last Track()
	fTrackDec		: LREAL;
	nSlew			: INT;		// number of Slew() calls
	fSlewAz			: LREAL;	// arguments of the last Slew()
	fSlewAlt		: LREAL;
	nOther			: INT;		// Home / Init / Park / Reset / Stop calls
END_VAR
VAR
	bCoverAutoOpen	: BOOL;
END_VAR

METHOD ClearCounters : BOOL
VAR_INPUT
END_VAR
nTrack := 0; fTrackRa := 0.0; fTrackDec := 0.0;
nSlew := 0; fSlewAz := 0.0; fSlewAlt := 0.0;
nOther := 0;
ClearCounters := TRUE;
END_METHOD

METHOD Home : BOOL
VAR_INPUT
END_VAR
nOther := nOther + 1;
Home := TRUE;
END_METHOD

METHOD Init : BOOL
VAR_INPUT
END_VAR
nOther := nOther + 1;
Init := TRUE;
END_METHOD

METHOD Park : BOOL
VAR_INPUT
END_VAR
nOther := nOther + 1;
Park := TRUE;
END_METHOD

METHOD Reset : BOOL
VAR_INPUT
END_VAR
nOther := nOther + 1;
Reset := TRUE;
END_METHOD

METHOD Stop : BOOL
VAR_INPUT
END_VAR
nOther := nOther + 1;
Stop := TRUE;
END_METHOD

METHOD Slew : BOOL
VAR_INPUT
	fAzimuth	: LREAL;
	fAltitude	: LREAL;
END_VAR
nSlew := nSlew + 1;
fSlewAz := fAzimuth;
fSlewAlt := fAltitude;
Slew := TRUE;
END_METHOD

METHOD Track : BOOL
VAR_INPUT
	fRightAscension	: LREAL;
	fDeclination	: LREAL;
END_VAR
nTrack := nTrack + 1;
fTrackRa := fRightAscension;
fTrackDec := fDeclination;
Track := TRUE;
END_METHOD

PROPERTY Altitude : LREAL
GET
Altitude := fSlewAlt;
END_GET
END_PROPERTY

PROPERTY Azimuth : LREAL
GET
Azimuth := fSlewAz;
END_GET
END_PROPERTY

PROPERTY Declination : LREAL
GET
Declination := fTrackDec;
END_GET
END_PROPERTY

PROPERTY RightAscension : LREAL
GET
RightAscension := fTrackRa;
END_GET
END_PROPERTY

PROPERTY CoverAutoOpen : BOOL
GET
CoverAutoOpen := bCoverAutoOpen;
END_GET
SET
bCoverAutoOpen := CoverAutoOpen;
END_SET
END_PROPERTY

END_FUNCTION_BLOCK

// ---- POUs/FB_InfoConnection_Tests.TcPOU
// Tests for BROTLib.FB_InfoConnection, the TwinSAFE connection diagnostics decoder (#12).
FUNCTION_BLOCK FB_InfoConnection_Tests EXTENDS TcUnit.FB_TestSuite
VAR
	fbInfo	: BROTLib.FB_InfoConnection;
END_VAR

No_Error();
Decodes_Every_Code();
Unknown_Codes();
Flags_Without_Code();
Code_And_Flags();
States();

// Runs fbInfo with usiMapDiag := nDiag and asserts sDiag = sExpected.
METHOD PRIVATE Check
VAR_INPUT
	nDiag		: USINT;
	sExpected	: STRING(255);
END_VAR
VAR
	stData		: BROTLib.ST_InfoDataConnection;
END_VAR
stData.usiMapDiag := nDiag;
fbInfo(stInfoData := stData);
AssertEquals_STRING(
	Expected := sExpected,
	Actual := fbInfo.sDiag,
	Message := CONCAT('sDiag for usiMapDiag = ', USINT_TO_STRING(nDiag)));
END_METHOD

METHOD PRIVATE No_Error
TEST('No_Error');
Check(nDiag := 0, sExpected := 'No error');
AssertEquals_USINT(Expected := 0, Actual := fbInfo.nDiagCode, Message := 'nDiagCode');
TEST_FINISHED();
END_METHOD

METHOD PRIVATE Decodes_Every_Code
VAR
	aTexts	: ARRAY[1..12] OF STRING := ['Invalid Command', 'Unknown Command', 'Invalid Connection ID', 'Invalid CRC', 'Watchdog expired', 'Invalid FSoE address', 'Invalid data', 'Invalid Com.-Parameter length', 'Invalid Com.-Parameter', 'Invalid User-Parameter length', 'Invalid User-Parameter', 'FSoE Master Reset'];
	i		: INT;
END_VAR
TEST('Decodes_Every_Code');
// 3, 5, 6, 7, 9, 10 and 11 decoded to 'Invalid Command' or 'Unknown Command' before #12
FOR i := 1 TO 12 DO
	Check(nDiag := INT_TO_USINT(i), sExpected := aTexts[i]);
	AssertEquals_USINT(Expected := INT_TO_USINT(i), Actual := fbInfo.nDiagCode, Message := aTexts[i]);
END_FOR
TEST_FINISHED();
END_METHOD

METHOD PRIVATE Unknown_Codes
TEST('Unknown_Codes');
Check(nDiag := 13, sExpected := 'Unknown error code 13');
Check(nDiag := 15, sExpected := 'Unknown error code 15');
TEST_FINISHED();
END_METHOD

METHOD PRIVATE Flags_Without_Code
TEST('Flags_Without_Code');
Check(nDiag := 16#10, sExpected := 'Error by FSoE Slave detected');
AssertTrue(Condition := fbInfo.bSlaveError, Message := 'bSlaveError');
Check(nDiag := 16#40, sExpected := 'StartUp');
AssertTrue(Condition := fbInfo.bStartUp, Message := 'bStartUp');
AssertFalse(Condition := fbInfo.bSlaveError, Message := 'bSlaveError cleared');
Check(nDiag := 16#A0, sExpected := 'FSoE Slave reports Failsafe value active; FSoE Master reports Failsafe value active');
AssertTrue(Condition := fbInfo.bSlaveFailsafe AND fbInfo.bMasterFailsafe, Message := 'failsafe flags');
TEST_FINISHED();
END_METHOD

METHOD PRIVATE Code_And_Flags
TEST('Code_And_Flags');
// before #12 any set low bit hid the flags
Check(nDiag := 16#15, sExpected := 'Watchdog expired; Error by FSoE Slave detected');
Check(nDiag := 16#FC, sExpected := 'FSoE Master Reset; Error by FSoE Slave detected; FSoE Slave reports Failsafe value active; StartUp; FSoE Master reports Failsafe value active');
AssertEquals_USINT(Expected := 12, Actual := fbInfo.nDiagCode, Message := 'nDiagCode');
TEST_FINISHED();
END_METHOD

METHOD PRIVATE States
VAR
	stData	: BROTLib.ST_InfoDataConnection;
END_VAR
TEST('States');
stData.usiMapState := 104;
fbInfo(stInfoData := stData);
AssertEquals_STRING(Expected := 'State Data', Actual := fbInfo.sState, Message := 'state 104');
stData.usiMapState := 7;
fbInfo(stInfoData := stData);
AssertEquals_STRING(Expected := 'Error', Actual := fbInfo.sState, Message := 'state 7');
TEST_FINISHED();
END_METHOD

END_FUNCTION_BLOCK

// ---- POUs/F_SetpointEnableExecute_Tests.TcPOU
// Tests for BROTLib.F_SetpointEnableExecute, FB_Axis's setpoint-enable Execute logic (#9). Each call is one cycle.
FUNCTION_BLOCK F_SetpointEnableExecute_Tests EXTENDS TcUnit.FB_TestSuite
VAR
END_VAR

Normal_Track();
Busy_Keeps_Execute();
Error_Drops_Execute_And_Holds_Off();
Reset_Rearms();
End_Of_Track_Rearms();
Error_With_Reset_Drops_First();

// Request sets Execute; once the block is done and the request has ended, Execute drops.
METHOD PRIVATE Normal_Track
VAR
	bFailed	: BOOL;
	bExecute	: BOOL;
END_VAR
TEST('Normal_Track');
bExecute := BROTLib.F_SetpointEnableExecute(Request := TRUE, Tracking := TRUE, Reset := FALSE, Execute := bExecute, Busy := FALSE, Done := FALSE, Error := FALSE, Failed := bFailed);
AssertEquals_BOOL(Expected := TRUE, Actual := bExecute, Message := 'request: Execute');
bExecute := BROTLib.F_SetpointEnableExecute(Request := TRUE, Tracking := TRUE, Reset := FALSE, Execute := bExecute, Busy := FALSE, Done := TRUE, Error := FALSE, Failed := bFailed);
AssertEquals_BOOL(Expected := TRUE, Actual := bExecute, Message := 'done, still requested: Execute');
bExecute := BROTLib.F_SetpointEnableExecute(Request := FALSE, Tracking := FALSE, Reset := FALSE, Execute := bExecute, Busy := FALSE, Done := TRUE, Error := FALSE, Failed := bFailed);
AssertEquals_BOOL(Expected := FALSE, Actual := bExecute, Message := 'request ended, done: Execute');
AssertEquals_BOOL(Expected := FALSE, Actual := bFailed, Message := 'never failed: Failed');
TEST_FINISHED();
END_METHOD

// The request ends while the block is busy: Execute stays until it is done.
METHOD PRIVATE Busy_Keeps_Execute
VAR
	bFailed	: BOOL;
	bExecute	: BOOL;
END_VAR
TEST('Busy_Keeps_Execute');
bExecute := BROTLib.F_SetpointEnableExecute(Request := TRUE, Tracking := TRUE, Reset := FALSE, Execute := bExecute, Busy := FALSE, Done := FALSE, Error := FALSE, Failed := bFailed);
bExecute := BROTLib.F_SetpointEnableExecute(Request := FALSE, Tracking := FALSE, Reset := FALSE, Execute := bExecute, Busy := TRUE, Done := FALSE, Error := FALSE, Failed := bFailed);
AssertEquals_BOOL(Expected := TRUE, Actual := bExecute, Message := 'busy: Execute');
bExecute := BROTLib.F_SetpointEnableExecute(Request := FALSE, Tracking := FALSE, Reset := FALSE, Execute := bExecute, Busy := FALSE, Done := TRUE, Error := FALSE, Failed := bFailed);
AssertEquals_BOOL(Expected := FALSE, Actual := bExecute, Message := 'done: Execute');
TEST_FINISHED();
END_METHOD

// The #9 latch: before, Execute stayed TRUE after an error and the axis could never track again.
METHOD PRIVATE Error_Drops_Execute_And_Holds_Off
VAR
	bFailed	: BOOL;
	bExecute	: BOOL;
END_VAR
TEST('Error_Drops_Execute_And_Holds_Off');
bExecute := BROTLib.F_SetpointEnableExecute(Request := TRUE, Tracking := TRUE, Reset := FALSE, Execute := bExecute, Busy := FALSE, Done := FALSE, Error := FALSE, Failed := bFailed);
bExecute := BROTLib.F_SetpointEnableExecute(Request := TRUE, Tracking := TRUE, Reset := FALSE, Execute := bExecute, Busy := FALSE, Done := FALSE, Error := TRUE, Failed := bFailed);
AssertEquals_BOOL(Expected := FALSE, Actual := bExecute, Message := 'error: Execute');
AssertEquals_BOOL(Expected := TRUE, Actual := bFailed, Message := 'error: Failed');
bExecute := BROTLib.F_SetpointEnableExecute(Request := TRUE, Tracking := TRUE, Reset := FALSE, Execute := bExecute, Busy := FALSE, Done := FALSE, Error := FALSE, Failed := bFailed);
AssertEquals_BOOL(Expected := FALSE, Actual := bExecute, Message := 'error cleared, still requested: no retry: Execute');
AssertEquals_BOOL(Expected := TRUE, Actual := bFailed, Message := 'still held off: Failed');
TEST_FINISHED();
END_METHOD

METHOD PRIVATE Reset_Rearms
VAR
	bFailed	: BOOL;
	bExecute	: BOOL;
END_VAR
TEST('Reset_Rearms');
bExecute := BROTLib.F_SetpointEnableExecute(Request := TRUE, Tracking := TRUE, Reset := FALSE, Execute := bExecute, Busy := FALSE, Done := FALSE, Error := FALSE, Failed := bFailed);
bExecute := BROTLib.F_SetpointEnableExecute(Request := TRUE, Tracking := TRUE, Reset := FALSE, Execute := bExecute, Busy := FALSE, Done := FALSE, Error := TRUE, Failed := bFailed);
bExecute := BROTLib.F_SetpointEnableExecute(Request := TRUE, Tracking := TRUE, Reset := TRUE, Execute := bExecute, Busy := FALSE, Done := FALSE, Error := FALSE, Failed := bFailed);
AssertEquals_BOOL(Expected := TRUE, Actual := bExecute, Message := 'reset: rising edge again: Execute');
AssertEquals_BOOL(Expected := FALSE, Actual := bFailed, Message := 'reset: Failed');
TEST_FINISHED();
END_METHOD

METHOD PRIVATE End_Of_Track_Rearms
VAR
	bFailed	: BOOL;
	bExecute	: BOOL;
END_VAR
TEST('End_Of_Track_Rearms');
bExecute := BROTLib.F_SetpointEnableExecute(Request := TRUE, Tracking := TRUE, Reset := FALSE, Execute := bExecute, Busy := FALSE, Done := FALSE, Error := FALSE, Failed := bFailed);
bExecute := BROTLib.F_SetpointEnableExecute(Request := TRUE, Tracking := TRUE, Reset := FALSE, Execute := bExecute, Busy := FALSE, Done := FALSE, Error := TRUE, Failed := bFailed);
bExecute := BROTLib.F_SetpointEnableExecute(Request := FALSE, Tracking := FALSE, Reset := FALSE, Execute := bExecute, Busy := FALSE, Done := FALSE, Error := FALSE, Failed := bFailed);
AssertEquals_BOOL(Expected := FALSE, Actual := bExecute, Message := 'track ended: Execute');
AssertEquals_BOOL(Expected := FALSE, Actual := bFailed, Message := 'track ended: Failed');
bExecute := BROTLib.F_SetpointEnableExecute(Request := TRUE, Tracking := TRUE, Reset := FALSE, Execute := bExecute, Busy := FALSE, Done := FALSE, Error := FALSE, Failed := bFailed);
AssertEquals_BOOL(Expected := TRUE, Actual := bExecute, Message := 'new track request: Execute');
TEST_FINISHED();
END_METHOD

// Error and Reset in the same cycle: Execute still drops once, so the next enable is a rising edge.
METHOD PRIVATE Error_With_Reset_Drops_First
VAR
	bFailed	: BOOL;
	bExecute	: BOOL;
END_VAR
TEST('Error_With_Reset_Drops_First');
bExecute := BROTLib.F_SetpointEnableExecute(Request := TRUE, Tracking := TRUE, Reset := FALSE, Execute := bExecute, Busy := FALSE, Done := FALSE, Error := FALSE, Failed := bFailed);
bExecute := BROTLib.F_SetpointEnableExecute(Request := TRUE, Tracking := TRUE, Reset := TRUE, Execute := bExecute, Busy := FALSE, Done := FALSE, Error := TRUE, Failed := bFailed);
AssertEquals_BOOL(Expected := FALSE, Actual := bExecute, Message := 'error and reset: Execute');
bExecute := BROTLib.F_SetpointEnableExecute(Request := TRUE, Tracking := TRUE, Reset := TRUE, Execute := bExecute, Busy := FALSE, Done := FALSE, Error := FALSE, Failed := bFailed);
AssertEquals_BOOL(Expected := TRUE, Actual := bExecute, Message := 'next cycle: Execute');
TEST_FINISHED();
END_METHOD

END_FUNCTION_BLOCK
